# B&R Automation Studio project Panasonic_LinkaPowerCP2_A2021055 (part 44)

#### Main.st - Init, cyclic, exit code
```iecst
PROGRAM _INIT
	(* Insert code here *)
	SKTcpClientTrace_1.Params.IPportClient := 19000;
	SKTcpClientTrace_1.Cmd.LoggerOn:= FALSE;
END_PROGRAM

PROGRAM _CYCLIC

	//Priradenie indexu paletky//
    a:= P3_StoperSrobovania.PAR.CisloPaletky;
	P3_StoperSrobovania.PAR.CisloPaletky_STRING:= USINT_TO_STRING(a);

    //Parametre komunikácie//
    memcpy(ADR(SKTcpClientTrace_1.Params.IPaddrServ),ADR('192.168.128.250'),SIZEOF('192.168.128.250'));

    SKTcpClientTrace_1.Params.IPportServ := 12000;

	SKTcpClientTrace_1.pDevice := ADR('HDD_LOGGER');
	SKTcpClientTrace_1.pFile := ADR('logger_sktcpclienttrace_7.log');
    SKTcpClientTrace_1();

    //Parametre komunikácie//
    //Vstupy pre server//
    SKTcpClientTrace_1.Params.Packet.type := TRCB_P3_Srobovanie_ST7.INPUTS.TYP_Prikazu;
    SKTcpClientTrace_1.Params.Packet.workplace := TRCB_P3_Srobovanie_ST7.INPUTS.CisloStanice;
    SKTcpClientTrace_1.Params.Packet.rfid := TRCB_P3_Srobovanie_ST7.INPUTS.CisloPaletky;
    SKTcpClientTrace_1.Params.Packet.master := TRCB_P3_Srobovanie_ST7.INPUTS.QRkodPowerCP;
    SKTcpClientTrace_1.Params.Packet.dps1:= TRCB_P3_Srobovanie_ST7.INPUTS.QRkodFiltra;
    SKTcpClientTrace_1.Params.Packet.dps2:= '';
    SKTcpClientTrace_1.Params.Packet.dps3:= '';
    SKTcpClientTrace_1.Params.Packet.dps4:= '';
    SKTcpClientTrace_1.Params.Packet.dps5:= '';
    SKTcpClientTrace_1.Params.Packet.operator_id := TRCB_P3_Srobovanie_ST7.INPUTS.ID_Operatora;
    SKTcpClientTrace_1.Params.Packet.data_report:= TRCB_P3_Srobovanie_ST7.INPUTS.Report;
    SKTcpClientTrace_1.Params.Packet.result := TRCB_P3_Srobovanie_ST7.INPUTS.StavPaletky;

    //Výstupy zo servera//
    TRCB_P3_Srobovanie_ST7.OUTPUTS.TYP_Prikazu:= SKTcpClientTrace_1.Internal.Splitter.out[1];
    TRCB_P3_Srobovanie_ST7.OUTPUTS.CisloStanice:= SKTcpClientTrace_1.Internal.Splitter.out[2];
    TRCB_P3_Srobovanie_ST7.OUTPUTS.CisloPaletky:= SKTcpClientTrace_1.Internal.Splitter.out[3];
    IF TRCB_P3_Srobovanie_ST7.INPUTS.TYP_Prikazu = '0' THEN
        TRCB_P3_Srobovanie_ST7.OUTPUTS.CisloEtikety:= SKTcpClientTrace_1.Internal.Splitter.out[4];
    ELSE
        TRCB_P3_Srobovanie_ST7.OUTPUTS.QRkodPowerCP:= SKTcpClientTrace_1.Internal.Splitter.out[4];
    END_IF
    TRCB_P3_Srobovanie_ST7.OUTPUTS.QRkodFiltra:= SKTcpClientTrace_1.Internal.Splitter.out[5];
    TRCB_P3_Srobovanie_ST7.OUTPUTS.ID_Operatora:= SKTcpClientTrace_1.Internal.Splitter.out[10];
    TRCB_P3_Srobovanie_ST7.OUTPUTS.DruhCinnostiNaPaletke:= SKTcpClientTrace_1.Internal.Splitter.out[11];
    TRCB_P3_Srobovanie_ST7.OUTPUTS.PovolenieCinnostiNaPaletke:= SKTcpClientTrace_1.Internal.Splitter.out[12];

    //Volanie funkcie SequenceControl//
    SequenceControl(SC:= SC_KOM_Server);

    CASE SC_KOM_Server.Step OF

        0:
            SC_KOM_Server.StepName:= '0 - Nulovanie';
            SKTcpClientTrace_1.Cmd.Send:= FALSE;
            TRCB_P3_Srobovanie_ST7.CMD.VyziadajStavPaletky_TYP1:= FALSE;
            TRCB_P3_Srobovanie_ST7.CMD.PriradQRkodFiltra_TYP3:= FALSE;
            TRCB_P3_Srobovanie_ST7.CMD.VyziadajCisloEtikety_TYP0:= FALSE;
            TRCB_P3_Srobovanie_ST7.CMD.OdosliStavPaletky_TYP2:= FALSE;
            TRCB_P3_Srobovanie_ST7.STATUS.KomunikaciaUkoncena:= FALSE;
			TRCB_P3_Srobovanie_ST7.STATUS.KomunikaciaError:= FALSE;
			TRCB_P3_Srobovanie_ST7.STATUS.KOM_READY:= FALSE;
            PocetDopytovNaServer:= 0;

            IF SKTcpClientTrace_1.Internal.Step = 0 THEN
                SKTcpClientTrace_1.Enable:= TRUE;
                SC_KOM_Server.ResetStep:= TRUE;
                SC_KOM_Server.Step:= 1;
            ELSIF SKTcpClientTrace_1.Internal.Step = 15 THEN
                SKTcpClientTrace_1.Enable:= TRUE;
                SC_KOM_Server.ResetStep:= TRUE;
                SC_KOM_Server.Step:= 1;
            ELSE
                SKTcpClientTrace_1.Enable:= FALSE;
            END_IF

        1:
            SC_KOM_Server.StepName:= '1 - Rozhodnutie o cinnosti';
            TRCB_P3_Srobovanie_ST7.STATUS.KOM_READY:= TRUE;
			IF TRCB_P3_Srobovanie_ST7.CMD.VyziadajStavPaletky_TYP1 THEN
                TRCB_P3_Srobovanie_ST7.STATUS.KOM_READY:= FALSE;
				SC_KOM_Server.Step:= 10;
            ELSIF TRCB_P3_Srobovanie_ST7.CMD.PriradQRkodFiltra_TYP3 THEN
                TRCB_P3_Srobovanie_ST7.STATUS.KOM_READY:= FALSE;
				SC_KOM_Server.Step:= 20;
            ELSIF TRCB_P3_Srobovanie_ST7.CMD.VyziadajCisloEtikety_TYP0 THEN
                TRCB_P3_Srobovanie_ST7.STATUS.KOM_READY:= FALSE;
				SC_KOM_Server.Step:= 30;
            ELSIF TRCB_P3_Srobovanie_ST7.CMD.OdosliStavPaletky_TYP2 THEN
				TRCB_P3_Srobovanie_ST7.STATUS.KOM_READY:= FALSE;
				SC_KOM_Server.Step:= 40;
			ELSIF TRCB_P3_Srobovanie_ST7.CMD.VyziadajStavPanatrace_TYP4 THEN
				TRCB_P3_Srobovanie_ST7.STATUS.KOM_READY:= FALSE;
				SC_KOM_Server.Step:= 50;
            END_IF

        10:
            SC_KOM_Server.StepName:= '10 - Vyziadanie stavu paletky - odoslanie dat na server';
            SC_KOM_Server.IdleTime.PT:= T#3s;
            SC_KOM_Server.AlarmTime.PT:= T#10s;
            SC_KOM_Server.AlarmTime.IN:= TRUE;

			TRCB_P3_Srobovanie_ST7.INPUTS.CisloPaletky:= 'Pal';
			brsstrcat(ADR(TRCB_P3_Srobovanie_ST7.INPUTS.CisloPaletky), ADR(P3_StoperSrobovania.PAR.CisloPaletky_STRING));

            TRCB_P3_Srobovanie_ST7.INPUTS.TYP_Prikazu:= '1';
            TRCB_P3_Srobovanie_ST7.INPUTS.CisloStanice:= 'ST7';
            TRCB_P3_Srobovanie_ST7.INPUTS.QRkodPowerCP:= Paletka[a].PAR.QRkodPowerCP;
            TRCB_P3_Srobovanie_ST7.INPUTS.QRkodFiltra:= '';
            TRCB_P3_Srobovanie_ST7.INPUTS.ID_Operatora:= Paletka[a].PAR.ID_Operatora;
            TRCB_P3_Srobovanie_ST7.INPUTS.Report:= '';
            TRCB_P3_Srobovanie_ST7.INPUTS.StavPaletky:= 'OK';

			IF SKTcpClientTrace_1.Status.staReadyToSend AND NOT SKTcpClientTrace_1.Cmd.Close THEN
				TRCB_P3_Srobovanie_ST7.OUTPUTS.TYP_Prikazu:= '';
				SKTcpClientTrace_1.Cmd.Send:= TRUE;
				SC_KOM_Server.ResetStep:= TRUE;
				SC_KOM_Server.Step:= 13;
			END_IF

		13:
            SC_KOM_Server.StepName:= '13 - Vyziadanie stavu paletky - odpoved servera';
            SC_KOM_Server.IdleTime.PT:= T#3s;
            SC_KOM_Server.AlarmTime.PT:= T#7s;
            SC_KOM_Server.AlarmTime.IN:= TRUE;

            IF SKTcpClientTrace_1.Status.staReceived AND
                (TRCB_P3_Srobovanie_ST7.OUTPUTS.TYP_Prikazu = TRCB_P3_Srobovanie_ST7.INPUTS.TYP_Prikazu) AND
                (TRCB_P3_Srobovanie_ST7.OUTPUTS.QRkodPowerCP = TRCB_P3_Srobovanie_ST7.INPUTS.QRkodPowerCP) THEN
                TRCB_P3_Srobovanie_ST7.STATUS.KomunikaciaUkoncena:= TRUE;
                SC_KOM_Server.ResetStep:= TRUE;
                SC_KOM_Server.Step:= 15;
            ELSIF SC_KOM_Server.AlarmTime.Q AND NOT SKTcpClientTrace_1.Status.staSending THEN
                PocetDopytovNaServer:= PocetDopytovNaServer + 1;
				SKTcpClientTrace_1.Cmd.Send:= FALSE;
				SKTcpClientTrace_1.Cmd.Close:= TRUE;
				SC_KOM_Server.ResetStep:= TRUE;
                SC_KOM_Server.Step:= 14;
            END_IF

        14:
            SC_KOM_Server.StepName:= '14 - Vyziadanie stavu paletky - cakam na opatovny dopyt na server';
            SC_KOM_Server.IdleTime.PT:= T#1s;
            SC_KOM_Server.AlarmTime.PT:= T#10s;
            SC_KOM_Server.IdleTime.IN:= TRUE;

            IF PocetDopytovNaServer < 3 THEN
                IF SC_KOM_Server.IdleTime.Q THEN
                    SC_KOM_Server.ResetStep:= TRUE;
                    SC_KOM_Server.Step:= 10;
                END_IF
            ELSE
                TRCB_P3_Srobovanie_ST7.STATUS.KomunikaciaError:= TRUE;
                SC_KOM_Server.ResetStep:= TRUE;
                SC_KOM_Server.Step:= 15;
            END_IF

        15:
            SC_KOM_Server.StepName:= '15 - Vyziadanie stavu paletky - cakam na ukoncenie komunikacie';
            SC_KOM_Server.IdleTime.PT:= T#3s;
            SC_KOM_Server.AlarmTime.PT:= T#10s;

            IF NOT TRCB_P3_Srobovanie_ST7.CMD.VyziadajStavPaletky_TYP1 THEN
                SC_KOM_Server.ResetStep:= TRUE;
                SC_KOM_Server.Step:= 0;
            END_IF

        20:
            SC_KOM_Server.StepName:= '20 - Priradenie QR kodu - odoslanie dat na server';
            SC_KOM_Server.IdleTime.PT:= T#3s;
            SC_KOM_Server.AlarmTime.PT:= T#10s;

            TRCB_P3_Srobovanie_ST7.INPUTS.TYP_Prikazu:= '3';
            TRCB_P3_Srobovanie_ST7.INPUTS.CisloStanice:= 'ST7';
            TRCB_P3_Srobovanie_ST7.INPUTS.CisloPaletky;
            TRCB_P3_Srobovanie_ST7.INPUTS.QRkodPowerCP:= Paletka[a].PAR.QRkodPowerCP;
            TRCB_P3_Srobovanie_ST7.INPUTS.QRkodFiltra:= '';
            TRCB_P3_Srobovanie_ST7.INPUTS.ID_Operatora:= Paletka[a].PAR.ID_Operatora;
            TRCB_P3_Srobovanie_ST7.INPUTS.Report:= '';
            TRCB_P3_Srobovanie_ST7.INPUTS.StavPaletky:= 'OK';
            SKTcpClientTrace_1.Cmd.Send:= TRUE;

            IF SKTcpClientTrace_1.Cmd.Send AND NOT SKTcpClientTrace_1.Status.staReceived AND NOT SKTcpClientTrace_1.Status.staError THEN
                SC_KOM_Server.ResetStep:= TRUE;
                SC_KOM_Server.Step:= 23;
            END_IF

        23:
            SC_KOM_Server.StepName:= '23 - Priradenie QR kodu - odpoved servera';
            SC_KOM_Server.IdleTime.PT:= T#3s;
            SC_KOM_Server.AlarmTime.PT:= T#20s;
            SC_KOM_Server.AlarmTime.IN:= TRUE;

            IF SKTcpClientTrace_1.Status.staReceived AND
                (TRCB_P3_Srobovanie_ST7.OUTPUTS.TYP_Prikazu = TRCB_P3_Srobovanie_ST7.INPUTS.TYP_Prikazu) AND
                (TRCB_P3_Srobovanie_ST7.OUTPUTS.QRkodPowerCP = TRCB_P3_Srobovanie_ST7.INPUTS.QRkodPowerCP) THEN
                TRCB_P3_Srobovanie_ST7.STATUS.KomunikaciaUkoncena:= TRUE;
                SC_KOM_Server.ResetStep:= TRUE;
                SC_KOM_Server.Step:= 25;
            ELSIF SC_KOM_Server.AlarmTime.Q THEN
                TRCB_P3_Srobovanie_ST7.STATUS.KomunikaciaError:= TRUE;
                SC_KOM_Server.ResetStep:= TRUE;
                SC_KOM_Server.Step:= 25;
            END_IF

        25:
            SC_KOM_Server.StepName:= '25 - Vyziadanie stavu paletky - cakam na ukoncenie komunikacie';
            SC_KOM_Server.IdleTime.PT:= T#3s;
            SC_KOM_Server.AlarmTime.PT:= T#10s;

            IF NOT TRCB_P3_Srobovanie_ST7.CMD.PriradQRkodFiltra_TYP3 THEN
                SC_KOM_Server.ResetStep:= TRUE;
                SC_KOM_Server.Step:= 0;
            END_IF

        30:
            SC_KOM_Server.StepName:= '30 - Vyziadanie serioveho cisla - odoslanie dat na server';
            SC_KOM_Server.IdleTime.PT:= T#3s;
            SC_KOM_Server.AlarmTime.PT:= T#10s;

            TRCB_P3_Srobovanie_ST7.INPUTS.TYP_Prikazu:= '0';
            TRCB_P3_Srobovanie_ST7.INPUTS.CisloStanice:= 'ST7';
            TRCB_P3_Srobovanie_ST7.INPUTS.CisloPaletky;
            TRCB_P3_Srobovanie_ST7.INPUTS.QRkodPowerCP:= '';
            TRCB_P3_Srobovanie_ST7.INPUTS.QRkodFiltra:= '';
            TRCB_P3_Srobovanie_ST7.INPUTS.ID_Operatora:= 'E2';
            TRCB_P3_Srobovanie_ST7.INPUTS.Report:= '';
            TRCB_P3_Srobovanie_ST7.INPUTS.StavPaletky:= 'OK';
            SKTcpClientTrace_1.Cmd.Send:= TRUE;

            IF SKTcpClientTrace_1.Cmd.Send AND NOT SKTcpClientTrace_1.Status.staReceived AND NOT SKTcpClientTrace_1.Status.staError THEN
                SC_KOM_Server.ResetStep:= TRUE;
                SC_KOM_Server.Step:= 33;
            END_IF

        33:
            SC_KOM_Server.StepName:= '33 - Vyziadanie serioveho cisla - odpoved servera';
            SC_KOM_Server.IdleTime.PT:= T#3s;
            SC_KOM_Server.AlarmTime.PT:= T#20s;
            SC_KOM_Server.AlarmTime.IN:= TRUE;

            IF SKTcpClientTrace_1.Status.staReceived AND
                (TRCB_P3_Srobovanie_ST7.OUTPUTS.TYP_Prikazu = TRCB_P3_Srobovanie_ST7.INPUTS.TYP_Prikazu) THEN
                TRCB_P3_Srobovanie_ST7.STATUS.KomunikaciaUkoncena:= TRUE;
                SC_KOM_Server.ResetStep:= TRUE;
                SC_KOM_Server.Step:= 35;
            ELSIF SC_KOM_Server.AlarmTime.Q THEN
                TRCB_P3_Srobovanie_ST7.STATUS.KomunikaciaError:= TRUE;
                SC_KOM_Server.ResetStep:= TRUE;
                SC_KOM_Server.Step:= 35;
            END_IF

        35:
            SC_KOM_Server.StepName:= '35 - Vyziadanie serioveho cisla - cakam na ukoncenie komunikacie';
            SC_KOM_Server.IdleTime.PT:= T#3s;
            SC_KOM_Server.AlarmTime.PT:= T#10s;

            IF NOT TRCB_P3_Srobovanie_ST7.CMD.VyziadajCisloEtikety_TYP0 THEN
                SC_KOM_Server.ResetStep:= TRUE;
                SC_KOM_Server.Step:= 0;
            END_IF

        40:
            SC_KOM_Server.StepName:= '40 - Odoslanie stavu paletky - odoslanie dat na server';
            SC_KOM_Server.IdleTime.PT:= T#3s;
            SC_KOM_Server.AlarmTime.PT:= T#20s;
            SC_KOM_Server.AlarmTime.IN:= TRUE;

            //Vytvorenie spravy pre report//
            IF NOT SC_KOM_Server.Switch1 THEN
                brsmemset(ADR(Report),0,SIZEOF(Report));
                brsmemset(ADR(TRCB_P3_Srobovanie_ST7.INPUTS.Report), 0, SIZEOF(TRCB_P3_Srobovanie_ST7.INPUTS.Report));

				//Skrutka K40//
                Report[0].PoradoveCislo:= '1';
                Report[0].Popis:= 'SkrutkaK40_Moment';
                Report[0].FormatHodnoty:= '1';
                Report[0].Tolerancia_MIN_Hodnota:= Reports.Skrutkovacky.Moment_ToleranciaMIN.P3_SkrutkaK40;
                Report[0].Tolerancia_MAX_Hodnota:= Reports.Skrutkovacky.Moment_ToleranciaMAX.P3_SkrutkaK40;
                Report[0].Nominal:= '';
                Report[0].Tolerancia_MIN_Jednotky:= 'Nm';
                Report[0].Tolerancia_MAX_Jednotky:= 'Nm';
                Report[0].NameranaHodnota:= Reports.Skrutkovacky.Moment_NameranaHodnota.P3_SkrutkaK40;
                Report[0].NameranaHodnota_Jednotky:= 'Nm';
                Report[0].VyslednyResult:= Reports.Skrutkovacky.VyslednyReport.P3_SkrutkaK40;
                SKTcpClientNewCsvEntry(Report[0].PoradoveCislo,Report[0].Popis,Report[0].FormatHodnoty,Report[0].Tolerancia_MIN_Hodnota,Report[0].Tolerancia_MAX_Hodnota,Report[0].Nominal,Report[0].Tolerancia_MIN_Jednotky,Report[0].Tolerancia_MAX_Jednotky,Report[0].NameranaHodnota,Report[0].NameranaHodnota_Jednotky,Report[0].VyslednyResult, ADR(TRCB_P3_Srobovanie_ST7.INPUTS.Report));

                Report[1].PoradoveCislo:= '2';
                Report[1].Popis:= 'SkrutkaK40_Uhol';
                Report[1].FormatHodnoty:= '1';
                Report[1].Tolerancia_MIN_Hodnota:= Reports.Skrutkovacky.Uhol_ToleranciaMIN.P3_SkrutkaK40;
                Report[1].Tolerancia_MAX_Hodnota:= Reports.Skrutkovacky.Uhol_ToleranciaMAX.P3_SkrutkaK40;
                Report[1].Nominal:= '';
                Report[1].Tolerancia_MIN_Jednotky:= 'st';
                Report[1].Tolerancia_MAX_Jednotky:= 'st';
                Report[1].NameranaHodnota:= Reports.Skrutkovacky.Uhol_NameranaHodnota.P3_SkrutkaK40;
                Report[1].NameranaHodnota_Jednotky:= 'st';
                Report[1].VyslednyResult:= Reports.Skrutkovacky.VyslednyReport.P3_SkrutkaK40;
                SKTcpClientNewCsvEntry(Report[1].PoradoveCislo,Report[1].Popis,Report[1].FormatHodnoty,Report[1].Tolerancia_MIN_Hodnota,Report[1].Tolerancia_MAX_Hodnota,Report[1].Nominal,Report[1].Tolerancia_MIN_Jednotky,Report[1].Tolerancia_MAX_Jednotky,Report[1].NameranaHodnota,Report[1].NameranaHodnota_Jednotky,Report[1].VyslednyResult, ADR(TRCB_P3_Srobovanie_ST7.INPUTS.Report));

                Report[2].PoradoveCislo:= '3';
                Report[2].Popis:= 'SkrutkaK40_CasSrobovania';
                Report[2].FormatHodnoty:= '1';
                Report[2].Tolerancia_MIN_Hodnota:= '';
                Report[2].Tolerancia_MAX_Hodnota:= '';
                Report[2].Nominal:= '';
                Report[2].Tolerancia_MIN_Jednotky:= '';
                Report[2].Tolerancia_MAX_Jednotky:= '';
                Report[2].NameranaHodnota:= Reports.Skrutkovacky.CasSkrutkovania.P3_SkrutkaK40;
                Report[2].NameranaHodnota_Jednotky:= 's';
                Report[2].VyslednyResult:= Reports.Skrutkovacky.VyslednyReport.P3_SkrutkaK40;
                SKTcpClientNewCsvEntry(Report[2].PoradoveCislo,Report[2].Popis,Report[2].FormatHodnoty,Report[2].Tolerancia_MIN_Hodnota,Report[2].Tolerancia_MAX_Hodnota,Report[2].Nominal,Report[2].Tolerancia_MIN_Jednotky,Report[2].Tolerancia_MAX_Jednotky,Report[2].NameranaHodnota,Report[2].NameranaHodnota_Jednotky,Report[2].VyslednyResult, ADR(TRCB_P3_Srobovanie_ST7.INPUTS.Report));

                Report[3].PoradoveCislo:= '4';
                Report[3].Popis:= 'SkrutkaK40_VyskaSrobovania';
                Report[3].FormatHodnoty:= '1';
                Report[3].Tolerancia_MIN_Hodnota:= '';
                Report[3].Tolerancia_MAX_Hodnota:= '';
                Report[3].Nominal:= '';
                Report[3].Tolerancia_MIN_Jednotky:= '';
                Report[3].Tolerancia_MAX_Jednotky:= '';
                Report[3].NameranaHodnota:= Reports.Skrutkovacky.VyskaSkrutkovania.P3_SkrutkaK40;
                Report[3].NameranaHodnota_Jednotky:= 'mm';
                Report[3].VyslednyResult:= Reports.Skrutkovacky.VyslednyReport.P3_SkrutkaK40;
                SKTcpClientNewCsvEntry(Report[3].PoradoveCislo,Report[3].Popis,Report[3].FormatHodnoty,Report[3].Tolerancia_MIN_Hodnota,Report[3].Tolerancia_MAX_Hodnota,Report[3].Nominal,Report[3].Tolerancia_MIN_Jednotky,Report[3].Tolerancia_MAX_Jednotky,Report[3].NameranaHodnota,Report[3].NameranaHodnota_Jednotky,Report[3].VyslednyResult, ADR(TRCB_P3_Srobovanie_ST7.INPUTS.Report));

                //Skrutka M5//
                Report[4].PoradoveCislo:= '5';
                Report[4].Popis:= 'SkrutkaM5_Moment';
                Report[4].FormatHodnoty:= '1';
                Report[4].Tolerancia_MIN_Hodnota:= Reports.Skrutkovacky.Moment_ToleranciaMIN.P3_SkrutkaM5;
                Report[4].Tolerancia_MAX_Hodnota:= Reports.Skrutkovacky.Moment_ToleranciaMAX.P3_SkrutkaM5;
                Report[4].Nominal:= '';
                Report[4].Tolerancia_MIN_Jednotky:= 'Nm';
                Report[4].Tolerancia_MAX_Jednotky:= 'Nm';
                Report[4].NameranaHodnota:= Reports.Skrutkovacky.Moment_NameranaHodnota.P3_SkrutkaM5;
                Report[4].NameranaHodnota_Jednotky:= 'Nm';
                Report[4].VyslednyResult:= Reports.Skrutkovacky.VyslednyReport.P3_SkrutkaM5;
                SKTcpClientNewCsvEntry(Report[4].PoradoveCislo,Report[4].Popis,Report[4].FormatHodnoty,Report[4].Tolerancia_MIN_Hodnota,Report[4].Tolerancia_MAX_Hodnota,Report[4].Nominal,Report[4].Tolerancia_MIN_Jednotky,Report[4].Tolerancia_MAX_Jednotky,Report[4].NameranaHodnota,Report[4].NameranaHodnota_Jednotky,Report[4].VyslednyResult, ADR(TRCB_P3_Srobovanie_ST7.INPUTS.Report));

                Report[5].PoradoveCislo:= '6';
                Report[5].Popis:= 'SkrutkaM5_Uhol';
                Report[5].FormatHodnoty:= '1';
                Report[5].Tolerancia_MIN_Hodnota:= Reports.Skrutkovacky.Uhol_ToleranciaMIN.P3_SkrutkaM5;
                Report[5].Tolerancia_MAX_Hodnota:= Reports.Skrutkovacky.Uhol_ToleranciaMAX.P3_SkrutkaM5;
                Report[5].Nominal:= '';
                Report[5].Tolerancia_MIN_Jednotky:= 'st';
                Report[5].Tolerancia_MAX_Jednotky:= 'st';
                Report[5].NameranaHodnota:= Reports.Skrutkovacky.Uhol_NameranaHodnota.P3_SkrutkaM5;
                Report[5].NameranaHodnota_Jednotky:= 'st';
                Report[5].VyslednyResult:= Reports.Skrutkovacky.VyslednyReport.P3_SkrutkaM5;
                SKTcpClientNewCsvEntry(Report[5].PoradoveCislo,Report[5].Popis,Report[5].FormatHodnoty,Report[5].Tolerancia_MIN_Hodnota,Report[5].Tolerancia_MAX_Hodnota,Report[5].Nominal,Report[5].Tolerancia_MIN_Jednotky,Report[5].Tolerancia_MAX_Jednotky,Report[5].NameranaHodnota,Report[5].NameranaHodnota_Jednotky,Report[5].VyslednyResult, ADR(TRCB_P3_Srobovanie_ST7.INPUTS.Report));

                Report[6].PoradoveCislo:= '7';
                Report[6].Popis:= 'SkrutkaM5_CasSrobovania';
                Report[6].FormatHodnoty:= '1';
                Report[6].Tolerancia_MIN_Hodnota:= '';
                Report[6].Tolerancia_MAX_Hodnota:= '';
                Report[6].Nominal:= '';
                Report[6].Tolerancia_MIN_Jednotky:= '';
                Report[6].Tolerancia_MAX_Jednotky:= '';
                Report[6].NameranaHodnota:= Reports.Skrutkovacky.CasSkrutkovania.P3_SkrutkaM5;
                Report[6].NameranaHodnota_Jednotky:= 's';
                Report[6].VyslednyResult:= Reports.Skrutkovacky.VyslednyReport.P3_SkrutkaM5;
                SKTcpClientNewCsvEntry(Report[6].PoradoveCislo,Report[6].Popis,Report[6].FormatHodnoty,Report[6].Tolerancia_MIN_Hodnota,Report[6].Tolerancia_MAX_Hodnota,Report[6].Nominal,Report[6].Tolerancia_MIN_Jednotky,Report[6].Tolerancia_MAX_Jednotky,Report[6].NameranaHodnota,Report[6].NameranaHodnota_Jednotky,Report[6].VyslednyResult, ADR(TRCB_P3_Srobovanie_ST7.INPUTS.Report));

                Report[7].PoradoveCislo:= '8';
                Report[7].Popis:= 'SkrutkaM5_VyskaSrobovania';
                Report[7].FormatHodnoty:= '1';
                Report[7].Tolerancia_MIN_Hodnota:= '';
                Report[7].Tolerancia_MAX_Hodnota:= '';
                Report[7].Nominal:= '';
                Report[7].Tolerancia_MIN_Jednotky:= '';
                Report[7].Tolerancia_MAX_Jednotky:= '';
                Report[7].NameranaHodnota:= Reports.Skrutkovacky.VyskaSkrutkovania.P3_SkrutkaM5;
                Report[7].NameranaHodnota_Jednotky:= 'mm';
                Report[7].VyslednyResult:= Reports.Skrutkovacky.VyslednyReport.P3_SkrutkaM5;
                SKTcpClientNewCsvEntry(Report[7].PoradoveCislo,Report[7].Popis,Report[7].FormatHodnoty,Report[7].Tolerancia_MIN_Hodnota,Report[7].Tolerancia_MAX_Hodnota,Report[7].Nominal,Report[7].Tolerancia_MIN_Jednotky,Report[7].Tolerancia_MAX_Jednotky,Report[7].NameranaHodnota,Report[7].NameranaHodnota_Jednotky,Report[7].VyslednyResult, ADR(TRCB_P3_Srobovanie_ST7.INPUTS.Report));

//                //Kamera 13//
//                Report[8].PoradoveCislo:= '9';
//                Report[8].Popis:= 'KAM_13_KontrolaPaletky';
//                Report[8].FormatHodnoty:= '2';
//                Report[8].Tolerancia_MIN_Hodnota:= '';
//                Report[8].Tolerancia_MAX_Hodnota:= '';
//                Report[8].Nominal:= 'OK';
//                Report[8].Tolerancia_MIN_Jednotky:= '';
//                Report[8].Tolerancia_MAX_Jednotky:= '';
//                IF Reports.Kamery.P3_CAM13_KontrolaPaletky = 'PASS' THEN
//                    Report[8].NameranaHodnota:= 'OK';
//                ELSE
//                    Report[8].NameranaHodnota:= 'NG';
//                END_IF
//                Report[8].NameranaHodnota_Jednotky:= '';
//                Report[8].VyslednyResult:= Reports.Kamery.P3_CAM13_KontrolaPaletky;
//                SKTcpClientNewCsvEntry(Report[8].PoradoveCislo,Report[8].Popis,Report[8].FormatHodnoty,Report[8].Tolerancia_MIN_Hodnota,Report[8].Tolerancia_MAX_Hodnota,Report[8].Nominal,Report[8].Tolerancia_MIN_Jednotky,Report[8].Tolerancia_MAX_Jednotky,Report[8].NameranaHodnota,Report[8].NameranaHodnota_Jednotky,Report[8].VyslednyResult, ADR(TRCB_P3_Srobovanie_ST7.INPUTS.Report));
//
                SC_KOM_Server.Switch1:= TRUE;
            END_IF

			TRCB_P3_Srobovanie_ST7.INPUTS.CisloPaletky:= 'Pal';
			brsstrcat(ADR(TRCB_P3_Srobovanie_ST7.INPUTS.CisloPaletky), ADR(P3_StoperSrobovania.PAR.CisloPaletky_STRING));

            TRCB_P3_Srobovanie_ST7.INPUTS.TYP_Prikazu:= '2';
            TRCB_P3_Srobovanie_ST7.INPUTS.CisloStanice:= 'ST7';
            TRCB_P3_Srobovanie_ST7.INPUTS.QRkodPowerCP:= Paletka[a].PAR.QRkodPowerCP;
            TRCB_P3_Srobovanie_ST7.INPUTS.QRkodFiltra:= '';
            TRCB_P3_Srobovanie_ST7.INPUTS.ID_Operatora:= Paletka[a].PAR.ID_Operatora;
            TRCB_P3_Srobovanie_ST7.INPUTS.StavPaletky:= Paletka[a].PAR.StavPowerCP;

			IF SKTcpClientTrace_1.Status.staReadyToSend AND NOT SKTcpClientTrace_1.Cmd.Close THEN
				TRCB_P3_Srobovanie_ST7.OUTPUTS.TYP_Prikazu:= '';
				SKTcpClientTrace_1.Cmd.Send:= TRUE;
				SC_KOM_Server.ResetStep:= TRUE;
				SC_KOM_Server.Step:= 43;
			END_IF

        43:
            SC_KOM_Server.StepName:= '43 - Odoslanie stavu paletky - odpoved servera';
			SC_KOM_Server.IdleTime.PT:= T#3s;
            SC_KOM_Server.AlarmTime.PT:= T#7s;
            SC_KOM_Server.AlarmTime.IN:= TRUE;

            IF SKTcpClientTrace_1.Status.staReceived AND
                (TRCB_P3_Srobovanie_ST7.OUTPUTS.TYP_Prikazu = TRCB_P3_Srobovanie_ST7.INPUTS.TYP_Prikazu) AND
                (TRCB_P3_Srobovanie_ST7.OUTPUTS.QRkodPowerCP = TRCB_P3_Srobovanie_ST7.INPUTS.QRkodPowerCP) THEN
                TRCB_P3_Srobovanie_ST7.STATUS.KomunikaciaUkoncena:= TRUE;
                SC_KOM_Server.ResetStep:= TRUE;
                SC_KOM_Server.Step:= 45;
            ELSIF SC_KOM_Server.AlarmTime.Q AND NOT SKTcpClientTrace_1.Status.staSending THEN
                PocetDopytovNaServer:= PocetDopytovNaServer + 1;
				SKTcpClientTrace_1.Cmd.Send:= FALSE;
				SKTcpClientTrace_1.Cmd.Close:= TRUE;
				SC_KOM_Server.ResetStep:= TRUE;
                SC_KOM_Server.Step:= 44;
            END_IF

        44:
            SC_KOM_Server.StepName:= '44 - Odoslanie stavu paletky - cakam na opatovny dopyt na server';
            SC_KOM_Server.IdleTime.PT:= T#1s;
            SC_KOM_Server.AlarmTime.PT:= T#10s;
            SC_KOM_Server.IdleTime.IN:= TRUE;
            SKTcpClientTrace_1.Cmd.Send:= FALSE;

            IF PocetDopytovNaServer < 3 THEN
                IF SC_KOM_Server.IdleTime.Q THEN
                    SC_KOM_Server.ResetStep:= TRUE;
                    SC_KOM_Server.Step:= 40;
                END_IF
            ELSE
                TRCB_P3_Srobovanie_ST7.STATUS.KomunikaciaError:= TRUE;
                SC_KOM_Server.ResetStep:= TRUE;
                SC_KOM_Server.Step:= 45;
            END_IF

        45:
            SC_KOM_Server.StepName:= '45 - Vyziadanie serioveho cisla - cakam na ukoncenie komunikacie';
            SC_KOM_Server.IdleTime.PT:= T#3s;
            SC_KOM_Server.AlarmTime.PT:= T#10s;

            IF NOT TRCB_P3_Srobovanie_ST7.CMD.OdosliStavPaletky_TYP2 THEN
                SC_KOM_Server.ResetStep:= TRUE;
                SC_KOM_Server.Step:= 0;
            END_IF

		50:
			SC_KOM_Server.StepName:= '50 - Vyziadanie stavu Panatrace - odoslanie dat na server';
			SC_KOM_Server.IdleTime.PT:= T#3s;
			SC_KOM_Server.AlarmTime.PT:= T#10s;
			SC_KOM_Server.AlarmTime.IN:= TRUE;

			TRCB_P3_Srobovanie_ST7.INPUTS.TYP_Prikazu:= '4';
			TRCB_P3_Srobovanie_ST7.INPUTS.CisloStanice:= 'ST7';
			TRCB_P3_Srobovanie_ST7.INPUTS.CisloPaletky:= '';
			TRCB_P3_Srobovanie_ST7.INPUTS.QRkodPowerCP:= '';
			TRCB_P3_Srobovanie_ST7.INPUTS.QRkodFiltra:= '';
			TRCB_P3_Srobovanie_ST7.INPUTS.ID_Operatora:= '';
			TRCB_P3_Srobovanie_ST7.INPUTS.Report:= '';
			TRCB_P3_Srobovanie_ST7.INPUTS.StavPaletky:= '';

			IF SKTcpClientTrace_1.Status.staReadyToSend AND NOT SKTcpClientTrace_1.Cmd.Close THEN
				TRCB_P3_Srobovanie_ST7.OUTPUTS.TYP_Prikazu:= '';
				SKTcpClientTrace_1.Cmd.Send:= TRUE;
				SC_KOM_Server.ResetStep:= TRUE;
				SC_KOM_Server.Step:= 53;
			END_IF

		53:
			SC_KOM_Server.StepName:= '53 - Vyziadanie stavu paletky - odpoved servera';
			SC_KOM_Server.IdleTime.PT:= T#30s;
			SC_KOM_Server.AlarmTime.PT:= T#7s;
			SC_KOM_Server.AlarmTime.IN:= TRUE;

			IF SKTcpClientTrace_1.Status.staReceived AND TRCB_P3_Srobovanie_ST7.OUTPUTS.TYP_Prikazu = TRCB_P3_Srobovanie_ST7.INPUTS.TYP_Prikazu THEN
				TRCB_P3_Srobovanie_ST7.STATUS.KomunikaciaUkoncena:= TRUE;
				SC_KOM_Server.ResetStep:= TRUE;
				SC_KOM_Server.Step:= 55;
			ELSIF SC_KOM_Server.AlarmTime.Q AND NOT SKTcpClientTrace_1.Status.staSending THEN
				PocetDopytovNaServer:= PocetDopytovNaServer + 1;
				SKTcpClientTrace_1.Cmd.Send:= FALSE;
				SKTcpClientTrace_1.Cmd.Close:= TRUE;
				SC_KOM_Server.ResetStep:= TRUE;
				SC_KOM_Server.Step:= 54;
			END_IF

		54:
			SC_KOM_Server.StepName:= '54 - Vyziadanie stavu paletky - cakam na opatovny dopyt na server';
			SC_KOM_Server.IdleTime.PT:= T#1s;
			SC_KOM_Server.AlarmTime.PT:= T#10s;
			SC_KOM_Server.IdleTime.IN:= TRUE;

			IF PocetDopytovNaServer < 3 THEN
				IF SC_KOM_Server.IdleTime.Q THEN
					SC_KOM_Server.ResetStep:= TRUE;
					SC_KOM_Server.Step:= 50;
				END_IF
			ELSE
				TRCB_P3_Srobovanie_ST7.STATUS.KomunikaciaError:= TRUE;
				SC_KOM_Server.ResetStep:= TRUE;
				SC_KOM_Server.Step:= 55;
			END_IF

		55:
			SC_KOM_Server.StepName:= '55 - Vyziadanie stavu paletky - cakam na ukoncenie komunikacie';
			SC_KOM_Server.IdleTime.PT:= T#3s;
			SC_KOM_Server.AlarmTime.PT:= T#10s;

			IF NOT TRCB_P3_Srobovanie_ST7.CMD.VyziadajStavPanatrace_TYP4 THEN
				SC_KOM_Server.ResetStep:= TRUE;
				SC_KOM_Server.Step:= 0;
			END_IF

    END_CASE

END_PROGRAM

PROGRAM _EXIT
	(* Insert code here *)

END_PROGRAM
```

#### Types.typ - Local data types
```iecst
TYPE
	Report_typ : 	STRUCT
		PoradoveCislo : STRING[2]; (*IDstep - Poradové čislo reportu*)
		Popis : STRING[100]; (*Description - Popis*)
		FormatHodnoty : STRING[2]; (*TypValue - Format zaslané hodnoty  1- Číslo, 2 - Znak*)
		Tolerancia_MIN_Hodnota : STRING[10]; (*MinTol - Minimálna tolerancia meranej veličiny*)
		Tolerancia_MAX_Hodnota : STRING[10]; (*MaxTol - Maximálna tolerancia meranej veličiny*)
		Nominal : STRING[10]; (*Nom - Ak jezvolený formát string tak tu zadáme OK inak je prazdna*)
		Tolerancia_MIN_Jednotky : STRING[10]; (*MinEle - Jednotky minimálnej tolerancie veličiny*)
		Tolerancia_MAX_Jednotky : STRING[10]; (*MaxEle - Jednotky maximálnej tolerancie veličiny*)
		NameranaHodnota : STRING[10]; (*Value - Namerana hodnota veličiny, ak su kamery tak bude hodnota OK alebo NG*)
		NameranaHodnota_Jednotky : STRING[10]; (*ValEle - Jednotky nameranej veličiny*)
		VyslednyResult : STRING[5]; (*Result - Výsledný result  PASS, FAIL, SKIP*)
	END_STRUCT;
END_TYPE
```

#### Variables.var - Local variables
```iecst
VAR
	SC_KOM_Server : SequenceControlTyp;
	SKTcpClientTrace_1 : SKTcpClientTrace;
	a : USINT;
	Report : ARRAY[0..50] OF Report_typ;
	PocetDopytovNaServer : USINT;
END_VAR
```

### Program Logical/TracebilitySystem/P3_LeakageTestA_ST8A (IEC)

#### Main.st - Init, cyclic, exit code
```iecst
PROGRAM _INIT
	(* Insert code here *)
	SKTcpClientTrace_1.Params.IPportClient := 20000;
	SKTcpClientTrace_1.Cmd.LoggerOn:= FALSE;
END_PROGRAM

PROGRAM _CYCLIC

	//Priradenie indexu paletky//
    a:= P3_LeakageTestA.PAR.CisloPaletky;
	P3_LeakageTestA.PAR.CisloPaletky_STRING:= USINT_TO_STRING(a);

    //Parametre komunikácie//
    memcpy(ADR(SKTcpClientTrace_1.Params.IPaddrServ),ADR('192.168.128.250'),SIZEOF('192.168.128.250'));

    SKTcpClientTrace_1.Params.IPportServ := 12000;

	SKTcpClientTrace_1.pDevice := ADR('HDD_LOGGER');
	SKTcpClientTrace_1.pFile := ADR('logger_sktcpclienttrace_8A.log');
    SKTcpClientTrace_1();

    //Parametre komunikácie//
    //Vstupy pre server//
    SKTcpClientTrace_1.Params.Packet.type := TRCB_P3_LeakageTestA_ST8A.INPUTS.TYP_Prikazu;
    SKTcpClientTrace_1.Params.Packet.workplace := TRCB_P3_LeakageTestA_ST8A.INPUTS.CisloStanice;
    SKTcpClientTrace_1.Params.Packet.rfid := TRCB_P3_LeakageTestA_ST8A.INPUTS.CisloPaletky;
    SKTcpClientTrace_1.Params.Packet.master := TRCB_P3_LeakageTestA_ST8A.INPUTS.QRkodPowerCP;
    SKTcpClientTrace_1.Params.Packet.dps1:= TRCB_P3_LeakageTestA_ST8A.INPUTS.QRkodFiltra;
    SKTcpClientTrace_1.Params.Packet.dps2:= '';
    SKTcpClientTrace_1.Params.Packet.dps3:= '';
    SKTcpClientTrace_1.Params.Packet.dps4:= '';
    SKTcpClientTrace_1.Params.Packet.dps5:= '';
    SKTcpClientTrace_1.Params.Packet.operator_id := TRCB_P3_LeakageTestA_ST8A.INPUTS.ID_Operatora;
    SKTcpClientTrace_1.Params.Packet.data_report:= TRCB_P3_LeakageTestA_ST8A.INPUTS.Report;
    SKTcpClientTrace_1.Params.Packet.result := TRCB_P3_LeakageTestA_ST8A.INPUTS.StavPaletky;

    //Výstupy zo servera//
    TRCB_P3_LeakageTestA_ST8A.OUTPUTS.TYP_Prikazu:= SKTcpClientTrace_1.Internal.Splitter.out[1];
    TRCB_P3_LeakageTestA_ST8A.OUTPUTS.CisloStanice:= SKTcpClientTrace_1.Internal.Splitter.out[2];
    TRCB_P3_LeakageTestA_ST8A.OUTPUTS.CisloPaletky:= SKTcpClientTrace_1.Internal.Splitter.out[3];
    IF TRCB_P3_LeakageTestA_ST8A.INPUTS.TYP_Prikazu = '0' THEN
        TRCB_P3_LeakageTestA_ST8A.OUTPUTS.CisloEtikety:= SKTcpClientTrace_1.Internal.Splitter.out[4];
    ELSE
        TRCB_P3_LeakageTestA_ST8A.OUTPUTS.QRkodPowerCP:= SKTcpClientTrace_1.Internal.Splitter.out[4];
    END_IF
    TRCB_P3_LeakageTestA_ST8A.OUTPUTS.QRkodFiltra:= SKTcpClientTrace_1.Internal.Splitter.out[5];
    TRCB_P3_LeakageTestA_ST8A.OUTPUTS.ID_Operatora:= SKTcpClientTrace_1.Internal.Splitter.out[10];
    TRCB_P3_LeakageTestA_ST8A.OUTPUTS.DruhCinnostiNaPaletke:= SKTcpClientTrace_1.Internal.Splitter.out[11];
    TRCB_P3_LeakageTestA_ST8A.OUTPUTS.PovolenieCinnostiNaPaletke:= SKTcpClientTrace_1.Internal.Splitter.out[12];

    //Volanie funkcie SequenceControl//
    SequenceControl(SC:= SC_KOM_Server);

    CASE SC_KOM_Server.Step OF

        0:
            SC_KOM_Server.StepName:= '0 - Nulovanie';
            SKTcpClientTrace_1.Cmd.Send:= FALSE;
            TRCB_P3_LeakageTestA_ST8A.CMD.VyziadajStavPaletky_TYP1:= FALSE;
            TRCB_P3_LeakageTestA_ST8A.CMD.PriradQRkodFiltra_TYP3:= FALSE;
            TRCB_P3_LeakageTestA_ST8A.CMD.VyziadajCisloEtikety_TYP0:= FALSE;
			TRCB_P3_LeakageTestA_ST8A.CMD.OdosliStavPaletky_TYP2:= FALSE;
			TRCB_P3_LeakageTestA_ST8A.CMD.VyziadajStavPanatrace_TYP4:= FALSE;
            TRCB_P3_LeakageTestA_ST8A.STATUS.KomunikaciaUkoncena:= FALSE;
			TRCB_P3_LeakageTestA_ST8A.STATUS.KomunikaciaError:= FALSE;
			TRCB_P3_LeakageTestA_ST8A.STATUS.KOM_READY:= FALSE;
            PocetDopytovNaServer:= 0;

            IF SKTcpClientTrace_1.Internal.Step = 0 THEN
                SKTcpClientTrace_1.Enable:= TRUE;
                SC_KOM_Server.ResetStep:= TRUE;
                SC_KOM_Server.Step:= 1;
            ELSIF SKTcpClientTrace_1.Internal.Step = 15 THEN
                SKTcpClientTrace_1.Enable:= TRUE;
                SC_KOM_Server.ResetStep:= TRUE;
                SC_KOM_Server.Step:= 1;
            ELSE
                SKTcpClientTrace_1.Enable:= FALSE;
            END_IF

        1:
            SC_KOM_Server.StepName:= '1 - Rozhodnutie o cinnosti';
            TRCB_P3_LeakageTestA_ST8A.STATUS.KOM_READY:= TRUE;
			IF TRCB_P3_LeakageTestA_ST8A.CMD.VyziadajStavPaletky_TYP1 THEN
                TRCB_P3_LeakageTestA_ST8A.STATUS.KOM_READY:= FALSE;
				SC_KOM_Server.Step:= 10;
            ELSIF TRCB_P3_LeakageTestA_ST8A.CMD.PriradQRkodFiltra_TYP3 THEN
                TRCB_P3_LeakageTestA_ST8A.STATUS.KOM_READY:= FALSE;
				SC_KOM_Server.Step:= 20;
            ELSIF TRCB_P3_LeakageTestA_ST8A.CMD.VyziadajCisloEtikety_TYP0 THEN
                TRCB_P3_LeakageTestA_ST8A.STATUS.KOM_READY:= FALSE;
				SC_KOM_Server.Step:= 30;
            ELSIF TRCB_P3_LeakageTestA_ST8A.CMD.OdosliStavPaletky_TYP2 THEN
				TRCB_P3_LeakageTestA_ST8A.STATUS.KOM_READY:= FALSE;
				SC_KOM_Server.Step:= 40;
			ELSIF TRCB_P3_LeakageTestA_ST8A.CMD.VyziadajStavPanatrace_TYP4 THEN
				TRCB_P3_LeakageTestA_ST8A.STATUS.KOM_READY:= FALSE;
				SC_KOM_Server.Step:= 50;
            END_IF

        10:
            SC_KOM_Server.StepName:= '10 - Vyziadanie stavu paletky - odoslanie dat na server';
            SC_KOM_Server.IdleTime.PT:= T#3s;
            SC_KOM_Server.AlarmTime.PT:= T#10s;
            SC_KOM_Server.AlarmTime.IN:= TRUE;

			TRCB_P3_LeakageTestA_ST8A.INPUTS.CisloPaletky:= 'Pal';
			brsstrcat(ADR(TRCB_P3_LeakageTestA_ST8A.INPUTS.CisloPaletky), ADR(P3_LeakageTestA.PAR.CisloPaletky_STRING));

            TRCB_P3_LeakageTestA_ST8A.INPUTS.TYP_Prikazu:= '1';
            TRCB_P3_LeakageTestA_ST8A.INPUTS.CisloStanice:= 'ST8A';
            TRCB_P3_LeakageTestA_ST8A.INPUTS.QRkodPowerCP:= Paletka[a].PAR.QRkodPowerCP;
            TRCB_P3_LeakageTestA_ST8A.INPUTS.QRkodFiltra:= '';
            TRCB_P3_LeakageTestA_ST8A.INPUTS.ID_Operatora:= Paletka[a].PAR.ID_Operatora;
            TRCB_P3_LeakageTestA_ST8A.INPUTS.Report:= '';
            TRCB_P3_LeakageTestA_ST8A.INPUTS.StavPaletky:= 'OK';

			IF SKTcpClientTrace_1.Status.staReadyToSend AND NOT SKTcpClientTrace_1.Cmd.Close THEN
				TRCB_P3_LeakageTestA_ST8A.OUTPUTS.TYP_Prikazu:= '';
				SKTcpClientTrace_1.Cmd.Send:= TRUE;
				SC_KOM_Server.ResetStep:= TRUE;
				SC_KOM_Server.Step:= 13;
			END_IF

		13:
            SC_KOM_Server.StepName:= '13 - Vyziadanie stavu paletky - odpoved servera';
            SC_KOM_Server.IdleTime.PT:= T#3s;
            SC_KOM_Server.AlarmTime.PT:= T#7s;
            SC_KOM_Server.AlarmTime.IN:= TRUE;

            IF SKTcpClientTrace_1.Status.staReceived AND
                (TRCB_P3_LeakageTestA_ST8A.OUTPUTS.TYP_Prikazu = TRCB_P3_LeakageTestA_ST8A.INPUTS.TYP_Prikazu) AND
                (TRCB_P3_LeakageTestA_ST8A.OUTPUTS.QRkodPowerCP = TRCB_P3_LeakageTestA_ST8A.INPUTS.QRkodPowerCP) THEN
                TRCB_P3_LeakageTestA_ST8A.STATUS.KomunikaciaUkoncena:= TRUE;
                SC_KOM_Server.ResetStep:= TRUE;
                SC_KOM_Server.Step:= 15;
            ELSIF SC_KOM_Server.AlarmTime.Q AND NOT SKTcpClientTrace_1.Status.staSending THEN
                PocetDopytovNaServer:= PocetDopytovNaServer + 1;
				SKTcpClientTrace_1.Cmd.Send:= FALSE;
				SKTcpClientTrace_1.Cmd.Close:= TRUE;
				SC_KOM_Server.ResetStep:= TRUE;
                SC_KOM_Server.Step:= 14;
            END_IF

        14:
            SC_KOM_Server.StepName:= '14 - Vyziadanie stavu paletky - cakam na opatovny dopyt na server';
            SC_KOM_Server.IdleTime.PT:= T#1s;
            SC_KOM_Server.AlarmTime.PT:= T#10s;
            SC_KOM_Server.IdleTime.IN:= TRUE;

            IF PocetDopytovNaServer < 3 THEN
                IF SC_KOM_Server.IdleTime.Q THEN
                    SC_KOM_Server.ResetStep:= TRUE;
                    SC_KOM_Server.Step:= 10;
                END_IF
            ELSE
                TRCB_P3_LeakageTestA_ST8A.STATUS.KomunikaciaError:= TRUE;
                SC_KOM_Server.ResetStep:= TRUE;
                SC_KOM_Server.Step:= 15;
            END_IF

        15:
            SC_KOM_Server.StepName:= '15 - Vyziadanie stavu paletky - cakam na ukoncenie komunikacie';
            SC_KOM_Server.IdleTime.PT:= T#3s;
            SC_KOM_Server.AlarmTime.PT:= T#10s;

            IF NOT TRCB_P3_LeakageTestA_ST8A.CMD.VyziadajStavPaletky_TYP1 THEN
                SC_KOM_Server.ResetStep:= TRUE;
                SC_KOM_Server.Step:= 0;
            END_IF

        20:
            SC_KOM_Server.StepName:= '20 - Priradenie QR kodu - odoslanie dat na server';
            SC_KOM_Server.IdleTime.PT:= T#3s;
            SC_KOM_Server.AlarmTime.PT:= T#10s;

            TRCB_P3_LeakageTestA_ST8A.INPUTS.TYP_Prikazu:= '3';
            TRCB_P3_LeakageTestA_ST8A.INPUTS.CisloStanice:= 'ST8A';
            TRCB_P3_LeakageTestA_ST8A.INPUTS.CisloPaletky;
            TRCB_P3_LeakageTestA_ST8A.INPUTS.QRkodPowerCP:= Paletka[a].PAR.QRkodPowerCP;
            TRCB_P3_LeakageTestA_ST8A.INPUTS.QRkodFiltra:= '';
            TRCB_P3_LeakageTestA_ST8A.INPUTS.ID_Operatora:= Paletka[a].PAR.ID_Operatora;
            TRCB_P3_LeakageTestA_ST8A.INPUTS.Report:= '';
            TRCB_P3_LeakageTestA_ST8A.INPUTS.StavPaletky:= 'OK';
            SKTcpClientTrace_1.Cmd.Send:= TRUE;

            IF SKTcpClientTrace_1.Cmd.Send AND NOT SKTcpClientTrace_1.Status.staReceived AND NOT SKTcpClientTrace_1.Status.staError THEN
                SC_KOM_Server.ResetStep:= TRUE;
                SC_KOM_Server.Step:= 23;
            END_IF

        23:
            SC_KOM_Server.StepName:= '23 - Priradenie QR kodu - odpoved servera';
            SC_KOM_Server.IdleTime.PT:= T#3s;
            SC_KOM_Server.AlarmTime.PT:= T#20s;
            SC_KOM_Server.AlarmTime.IN:= TRUE;

            IF SKTcpClientTrace_1.Status.staReceived AND
                (TRCB_P3_LeakageTestA_ST8A.OUTPUTS.TYP_Prikazu = TRCB_P3_LeakageTestA_ST8A.INPUTS.TYP_Prikazu) AND
                (TRCB_P3_LeakageTestA_ST8A.OUTPUTS.QRkodPowerCP = TRCB_P3_LeakageTestA_ST8A.INPUTS.QRkodPowerCP) THEN
                TRCB_P3_LeakageTestA_ST8A.STATUS.KomunikaciaUkoncena:= TRUE;
                SC_KOM_Server.ResetStep:= TRUE;
                SC_KOM_Server.Step:= 25;
            ELSIF SC_KOM_Server.AlarmTime.Q THEN
                TRCB_P3_LeakageTestA_ST8A.STATUS.KomunikaciaError:= TRUE;
                SC_KOM_Server.ResetStep:= TRUE;
                SC_KOM_Server.Step:= 25;
            END_IF

        25:
            SC_KOM_Server.StepName:= '25 - Vyziadanie stavu paletky - cakam na ukoncenie komunikacie';
            SC_KOM_Server.IdleTime.PT:= T#3s;
            SC_KOM_Server.AlarmTime.PT:= T#10s;

            IF NOT TRCB_P3_LeakageTestA_ST8A.CMD.PriradQRkodFiltra_TYP3 THEN
                SC_KOM_Server.ResetStep:= TRUE;
                SC_KOM_Server.Step:= 0;
            END_IF

        30:
            SC_KOM_Server.StepName:= '30 - Vyziadanie serioveho cisla - odoslanie dat na server';
            SC_KOM_Server.IdleTime.PT:= T#3s;
            SC_KOM_Server.AlarmTime.PT:= T#10s;

            TRCB_P3_LeakageTestA_ST8A.INPUTS.TYP_Prikazu:= '0';
            TRCB_P3_LeakageTestA_ST8A.INPUTS.CisloStanice:= 'ST8A';
            TRCB_P3_LeakageTestA_ST8A.INPUTS.CisloPaletky;
            TRCB_P3_LeakageTestA_ST8A.INPUTS.QRkodPowerCP:= '';
            TRCB_P3_LeakageTestA_ST8A.INPUTS.QRkodFiltra:= '';
            TRCB_P3_LeakageTestA_ST8A.INPUTS.ID_Operatora:= 'E2';
            TRCB_P3_LeakageTestA_ST8A.INPUTS.Report:= '';
            TRCB_P3_LeakageTestA_ST8A.INPUTS.StavPaletky:= 'OK';
            SKTcpClientTrace_1.Cmd.Send:= TRUE;

            IF SKTcpClientTrace_1.Cmd.Send AND NOT SKTcpClientTrace_1.Status.staReceived AND NOT SKTcpClientTrace_1.Status.staError THEN
                SC_KOM_Server.ResetStep:= TRUE;
                SC_KOM_Server.Step:= 33;
            END_IF

        33:
            SC_KOM_Server.StepName:= '33 - Vyziadanie serioveho cisla - odpoved servera';
            SC_KOM_Server.IdleTime.PT:= T#3s;
            SC_KOM_Server.AlarmTime.PT:= T#20s;
            SC_KOM_Server.AlarmTime.IN:= TRUE;

            IF SKTcpClientTrace_1.Status.staReceived AND
                (TRCB_P3_LeakageTestA_ST8A.OUTPUTS.TYP_Prikazu = TRCB_P3_LeakageTestA_ST8A.INPUTS.TYP_Prikazu) THEN
                TRCB_P3_LeakageTestA_ST8A.STATUS.KomunikaciaUkoncena:= TRUE;
                SC_KOM_Server.ResetStep:= TRUE;
                SC_KOM_Server.Step:= 35;
            ELSIF SC_KOM_Server.AlarmTime.Q THEN
                TRCB_P3_LeakageTestA_ST8A.STATUS.KomunikaciaError:= TRUE;
                SC_KOM_Server.ResetStep:= TRUE;
                SC_KOM_Server.Step:= 35;
            END_IF

        35:
            SC_KOM_Server.StepName:= '35 - Vyziadanie serioveho cisla - cakam na ukoncenie komunikacie';
            SC_KOM_Server.IdleTime.PT:= T#3s;
            SC_KOM_Server.AlarmTime.PT:= T#10s;

            IF NOT TRCB_P3_LeakageTestA_ST8A.CMD.VyziadajCisloEtikety_TYP0 THEN
                SC_KOM_Server.ResetStep:= TRUE;
                SC_KOM_Server.Step:= 0;
            END_IF

        40:
            SC_KOM_Server.StepName:= '40 - Odoslanie stavu paletky - odoslanie dat na server';
            SC_KOM_Server.IdleTime.PT:= T#3s;
            SC_KOM_Server.AlarmTime.PT:= T#20s;
            SC_KOM_Server.AlarmTime.IN:= TRUE;

            //Vytvorenie spravy pre report//
            IF NOT SC_KOM_Server.Switch1 THEN
                brsmemset(ADR(Report),0,SIZEOF(Report));
                brsmemset(ADR(TRCB_P3_LeakageTestA_ST8A.INPUTS.Report), 0, SIZEOF(TRCB_P3_LeakageTestA_ST8A.INPUTS.Report));

				//Čas plnenia//
                Report[0].PoradoveCislo:= '1';
                Report[0].Popis:= 'StanicaA_CasPlnenia';
                Report[0].FormatHodnoty:= '1';
                Report[0].Tolerancia_MIN_Hodnota:= '';
                Report[0].Tolerancia_MAX_Hodnota:= '';
                Report[0].Nominal:= '';
                Report[0].Tolerancia_MIN_Jednotky:= '';
                Report[0].Tolerancia_MAX_Jednotky:= '';
                Report[0].NameranaHodnota:= Reports.LeakageTest.CasPlnenia.StanicaA;
                Report[0].NameranaHodnota_Jednotky:= 's';
                Report[0].VyslednyResult:= Reports.LeakageTest.VyslednyReport.StanicaA;
                SKTcpClientNewCsvEntry(Report[0].PoradoveCislo,Report[0].Popis,Report[0].FormatHodnoty,Report[0].Tolerancia_MIN_Hodnota,Report[0].Tolerancia_MAX_Hodnota,Report[0].Nominal,Report[0].Tolerancia_MIN_Jednotky,Report[0].Tolerancia_MAX_Jednotky,Report[0].NameranaHodnota,Report[0].NameranaHodnota_Jednotky,Report[0].VyslednyResult, ADR(TRCB_P3_LeakageTestA_ST8A.INPUTS.Report));

                //Čas stabilizacie//
                Report[1].PoradoveCislo:= '2';
                Report[1].Popis:= 'StanicaA_CasStabilizacie';
                Report[1].FormatHodnoty:= '1';
                Report[1].Tolerancia_MIN_Hodnota:= '';
                Report[1].Tolerancia_MAX_Hodnota:= '';
                Report[1].Nominal:= '';
                Report[1].Tolerancia_MIN_Jednotky:= '';
                Report[1].Tolerancia_MAX_Jednotky:= '';
                Report[1].NameranaHodnota:= Reports.LeakageTest.CasStabilizacie.StanicaA;
                Report[1].NameranaHodnota_Jednotky:= 's';
                Report[1].VyslednyResult:= Reports.LeakageTest.VyslednyReport.StanicaA;
                SKTcpClientNewCsvEntry(Report[1].PoradoveCislo,Report[1].Popis,Report[1].FormatHodnoty,Report[1].Tolerancia_MIN_Hodnota,Report[1].Tolerancia_MAX_Hodnota,Report[1].Nominal,Report[1].Tolerancia_MIN_Jednotky,Report[1].Tolerancia_MAX_Jednotky,Report[1].NameranaHodnota,Report[1].NameranaHodnota_Jednotky,Report[1].VyslednyResult, ADR(TRCB_P3_LeakageTestA_ST8A.INPUTS.Report));

                //Tlak plnenia//
                Report[2].PoradoveCislo:= '3';
                Report[2].Popis:= 'StanicaA_TlakPlnenia';
                Report[2].FormatHodnoty:= '1';
                Report[2].Tolerancia_MIN_Hodnota:= '';
                Report[2].Tolerancia_MAX_Hodnota:= '';
                Report[2].Nominal:= '';
                Report[2].Tolerancia_MIN_Jednotky:= '';
                Report[2].Tolerancia_MAX_Jednotky:= '';
                Report[2].NameranaHodnota:= Reports.LeakageTest.TlakPlnenia.StanicaA;
                Report[2].NameranaHodnota_Jednotky:= 'mBar';
                Report[2].VyslednyResult:= Reports.LeakageTest.VyslednyReport.StanicaA;
                SKTcpClientNewCsvEntry(Report[2].PoradoveCislo,Report[2].Popis,Report[2].FormatHodnoty,Report[2].Tolerancia_MIN_Hodnota,Report[2].Tolerancia_MAX_Hodnota,Report[2].Nominal,Report[2].Tolerancia_MIN_Jednotky,Report[2].Tolerancia_MAX_Jednotky,Report[2].NameranaHodnota,Report[2].NameranaHodnota_Jednotky,Report[2].VyslednyResult, ADR(TRCB_P3_LeakageTestA_ST8A.INPUTS.Report));

                //Tlak prítlaku//
                Report[3].PoradoveCislo:= '4';
                Report[3].Popis:= 'StanicaA_TlakPritlaku';
                Report[3].FormatHodnoty:= '1';
                Report[3].Tolerancia_MIN_Hodnota:= Reports.LeakageTest.ToleranciaPritlaku_MIN.StanicaA;
                Report[3].Tolerancia_MAX_Hodnota:= Reports.LeakageTest.ToleranciaPritlaku_MAX.StanicaA;
                Report[3].Nominal:= '';
                Report[3].Tolerancia_MIN_Jednotky:= 'Bar';
                Report[3].Tolerancia_MAX_Jednotky:= 'Bar';
                Report[3].NameranaHodnota:= Reports.LeakageTest.TlakPritlaku.StanicaA;
                Report[3].NameranaHodnota_Jednotky:= 'Bar';
                Report[3].VyslednyResult:= Reports.LeakageTest.VyslednyReport.StanicaA;
                SKTcpClientNewCsvEntry(Report[3].PoradoveCislo,Report[3].Popis,Report[3].FormatHodnoty,Report[3].Tolerancia_MIN_Hodnota,Report[3].Tolerancia_MAX_Hodnota,Report[3].Nominal,Report[3].Tolerancia_MIN_Jednotky,Report[3].Tolerancia_MAX_Jednotky,Report[3].NameranaHodnota,Report[3].NameranaHodnota_Jednotky,Report[3].VyslednyResult, ADR(TRCB_P3_LeakageTestA_ST8A.INPUTS.Report));

                //Tlak úniku//
                Report[4].PoradoveCislo:= '5';
                Report[4].Popis:= 'StanicaA_TlakUniku';
                Report[4].FormatHodnoty:= '1';
                Report[4].Tolerancia_MIN_Hodnota:= Reports.LeakageTest.ToleranciaTlakUniku_MIN.StanicaA;
                Report[4].Tolerancia_MAX_Hodnota:= Reports.LeakageTest.ToleranciaTlakUniku_MAX.StanicaA;
                Report[4].Nominal:= '';
                Report[4].Tolerancia_MIN_Jednotky:= 'Pa';
                Report[4].Tolerancia_MAX_Jednotky:= 'Pa';
                Report[4].NameranaHodnota:= Reports.LeakageTest.TlakUniku.StanicaA;
                Report[4].NameranaHodnota_Jednotky:= 'Pa';
                Report[4].VyslednyResult:= Reports.LeakageTest.VyslednyReport.StanicaA;
                SKTcpClientNewCsvEntry(Report[4].PoradoveCislo,Report[4].Popis,Report[4].FormatHodnoty,Report[4].Tolerancia_MIN_Hodnota,Report[4].Tolerancia_MAX_Hodnota,Report[4].Nominal,Report[4].Tolerancia_MIN_Jednotky,Report[4].Tolerancia_MAX_Jednotky,Report[4].NameranaHodnota,Report[4].NameranaHodnota_Jednotky,Report[4].VyslednyResult, ADR(TRCB_P3_LeakageTestA_ST8A.INPUTS.Report));

                //Tolerancia//
                Report[5].PoradoveCislo:= '6';
                Report[5].Popis:= 'StanicaA_Tolerancia';
                Report[5].FormatHodnoty:= '1';
                Report[5].Tolerancia_MIN_Hodnota:= '';
                Report[5].Tolerancia_MAX_Hodnota:= '';
                Report[5].Nominal:= '';
                Report[5].Tolerancia_MIN_Jednotky:= '';
                Report[5].Tolerancia_MAX_Jednotky:= '';
                Report[5].NameranaHodnota:= Reports.LeakageTest.Tolerancia.StanicaA;
                Report[5].NameranaHodnota_Jednotky:= 'Pa';
                Report[5].VyslednyResult:= Reports.LeakageTest.VyslednyReport.StanicaA;
                SKTcpClientNewCsvEntry(Report[5].PoradoveCislo,Report[5].Popis,Report[5].FormatHodnoty,Report[5].Tolerancia_MIN_Hodnota,Report[5].Tolerancia_MAX_Hodnota,Report[5].Nominal,Report[5].Tolerancia_MIN_Jednotky,Report[5].Tolerancia_MAX_Jednotky,Report[5].NameranaHodnota,Report[5].NameranaHodnota_Jednotky,Report[5].VyslednyResult, ADR(TRCB_P3_LeakageTestA_ST8A.INPUTS.Report));

                SC_KOM_Server.Switch1:= TRUE;
            END_IF

			TRCB_P3_LeakageTestA_ST8A.INPUTS.CisloPaletky:= 'Pal';
			brsstrcat(ADR(TRCB_P3_LeakageTestA_ST8A.INPUTS.CisloPaletky), ADR(P3_LeakageTestA.PAR.CisloPaletky_STRING));

            TRCB_P3_LeakageTestA_ST8A.INPUTS.TYP_Prikazu:= '2';
            TRCB_P3_LeakageTestA_ST8A.INPUTS.CisloStanice:= 'ST8A';
            TRCB_P3_LeakageTestA_ST8A.INPUTS.QRkodPowerCP:= Paletka[a].PAR.QRkodPowerCP;
            TRCB_P3_LeakageTestA_ST8A.INPUTS.QRkodFiltra:= '';
            TRCB_P3_LeakageTestA_ST8A.INPUTS.ID_Operatora:= Paletka[a].PAR.ID_Operatora;
            TRCB_P3_LeakageTestA_ST8A.INPUTS.StavPaletky:= Paletka[a].PAR.StavPowerCP;

			IF SKTcpClientTrace_1.Status.staReadyToSend AND NOT SKTcpClientTrace_1.Cmd.Close THEN
				TRCB_P3_LeakageTestA_ST8A.OUTPUTS.TYP_Prikazu:= '';
				SKTcpClientTrace_1.Cmd.Send:= TRUE;
				SC_KOM_Server.ResetStep:= TRUE;
				SC_KOM_Server.Step:= 43;
			END_IF

        43:
            SC_KOM_Server.StepName:= '43 - Odoslanie stavu paletky - odpoved servera';
			SC_KOM_Server.IdleTime.PT:= T#3s;
            SC_KOM_Server.AlarmTime.PT:= T#7s;
            SC_KOM_Server.AlarmTime.IN:= TRUE;

            IF SKTcpClientTrace_1.Status.staReceived AND
                (TRCB_P3_LeakageTestA_ST8A.OUTPUTS.TYP_Prikazu = TRCB_P3_LeakageTestA_ST8A.INPUTS.TYP_Prikazu) AND
                (TRCB_P3_LeakageTestA_ST8A.OUTPUTS.QRkodPowerCP = TRCB_P3_LeakageTestA_ST8A.INPUTS.QRkodPowerCP) THEN
                TRCB_P3_LeakageTestA_ST8A.STATUS.KomunikaciaUkoncena:= TRUE;
                SC_KOM_Server.ResetStep:= TRUE;
                SC_KOM_Server.Step:= 45;
            ELSIF SC_KOM_Server.AlarmTime.Q AND NOT SKTcpClientTrace_1.Status.staSending THEN
                PocetDopytovNaServer:= PocetDopytovNaServer + 1;
				SKTcpClientTrace_1.Cmd.Send:= FALSE;
				SKTcpClientTrace_1.Cmd.Close:= TRUE;
				SC_KOM_Server.ResetStep:= TRUE;
                SC_KOM_Server.Step:= 44;
            END_IF

        44:
            SC_KOM_Server.StepName:= '44 - Odoslanie stavu paletky - cakam na opatovny dopyt na server';
            SC_KOM_Server.IdleTime.PT:= T#1s;
            SC_KOM_Server.AlarmTime.PT:= T#10s;
            SC_KOM_Server.IdleTime.IN:= TRUE;
            SKTcpClientTrace_1.Cmd.Send:= FALSE;

            IF PocetDopytovNaServer < 3 THEN
                IF SC_KOM_Server.IdleTime.Q THEN
                    SC_KOM_Server.ResetStep:= TRUE;
                    SC_KOM_Server.Step:= 40;
                END_IF
            ELSE
                TRCB_P3_LeakageTestA_ST8A.STATUS.KomunikaciaError:= TRUE;
                SC_KOM_Server.ResetStep:= TRUE;
                SC_KOM_Server.Step:= 45;
            END_IF

        45:
            SC_KOM_Server.StepName:= '45 - Odoslanie stavu paletky - cakam na ukoncenie komunikacie';
            SC_KOM_Server.IdleTime.PT:= T#3s;
            SC_KOM_Server.AlarmTime.PT:= T#10s;

            IF NOT TRCB_P3_LeakageTestA_ST8A.CMD.OdosliStavPaletky_TYP2 THEN
                SC_KOM_Server.ResetStep:= TRUE;
                SC_KOM_Server.Step:= 0;
            END_IF

		50:
			SC_KOM_Server.StepName:= '50 - Vyziadanie stavu Panatrace - odoslanie dat na server';
			SC_KOM_Server.IdleTime.PT:= T#3s;
			SC_KOM_Server.AlarmTime.PT:= T#10s;
			SC_KOM_Server.AlarmTime.IN:= TRUE;

			TRCB_P3_LeakageTestA_ST8A.INPUTS.TYP_Prikazu:= '4';
			TRCB_P3_LeakageTestA_ST8A.INPUTS.CisloStanice:= 'ST8A';
			TRCB_P3_LeakageTestA_ST8A.INPUTS.CisloPaletky:= '';
			TRCB_P3_LeakageTestA_ST8A.INPUTS.QRkodPowerCP:= '';
			TRCB_P3_LeakageTestA_ST8A.INPUTS.QRkodFiltra:= '';
			TRCB_P3_LeakageTestA_ST8A.INPUTS.ID_Operatora:= '';
			TRCB_P3_LeakageTestA_ST8A.INPUTS.Report:= '';
			TRCB_P3_LeakageTestA_ST8A.INPUTS.StavPaletky:= '';

			IF SKTcpClientTrace_1.Status.staReadyToSend AND NOT SKTcpClientTrace_1.Cmd.Close THEN
				TRCB_P3_LeakageTestA_ST8A.OUTPUTS.TYP_Prikazu:= '';
				SKTcpClientTrace_1.Cmd.Send:= TRUE;
				SC_KOM_Server.ResetStep:= TRUE;
				SC_KOM_Server.Step:= 53;
			END_IF

		53:
			SC_KOM_Server.StepName:= '53 - Vyziadanie stavu paletky - odpoved servera';
			SC_KOM_Server.IdleTime.PT:= T#30s;
			SC_KOM_Server.AlarmTime.PT:= T#7s;
			SC_KOM_Server.AlarmTime.IN:= TRUE;

			IF SKTcpClientTrace_1.Status.staReceived AND TRCB_P3_LeakageTestA_ST8A.OUTPUTS.TYP_Prikazu = TRCB_P3_LeakageTestA_ST8A.INPUTS.TYP_Prikazu THEN
				TRCB_P3_LeakageTestA_ST8A.STATUS.KomunikaciaUkoncena:= TRUE;
				SC_KOM_Server.ResetStep:= TRUE;
				SC_KOM_Server.Step:= 55;
			ELSIF SC_KOM_Server.AlarmTime.Q AND NOT SKTcpClientTrace_1.Status.staSending THEN
				PocetDopytovNaServer:= PocetDopytovNaServer + 1;
				SKTcpClientTrace_1.Cmd.Send:= FALSE;
				SKTcpClientTrace_1.Cmd.Close:= TRUE;
				SC_KOM_Server.ResetStep:= TRUE;
				SC_KOM_Server.Step:= 54;
			END_IF

		54:
			SC_KOM_Server.StepName:= '54 - Vyziadanie stavu paletky - cakam na opatovny dopyt na server';
			SC_KOM_Server.IdleTime.PT:= T#1s;
			SC_KOM_Server.AlarmTime.PT:= T#10s;
			SC_KOM_Server.IdleTime.IN:= TRUE;

			IF PocetDopytovNaServer < 3 THEN
				IF SC_KOM_Server.IdleTime.Q THEN
					SC_KOM_Server.ResetStep:= TRUE;
					SC_KOM_Server.Step:= 50;
				END_IF
			ELSE
				TRCB_P3_LeakageTestA_ST8A.STATUS.KomunikaciaError:= TRUE;
				SC_KOM_Server.ResetStep:= TRUE;
				SC_KOM_Server.Step:= 55;
			END_IF

		55:
			SC_KOM_Server.StepName:= '55 - Vyziadanie stavu paletky - cakam na ukoncenie komunikacie';
			SC_KOM_Server.IdleTime.PT:= T#3s;
			SC_KOM_Server.AlarmTime.PT:= T#10s;

			IF NOT TRCB_P3_LeakageTestA_ST8A.CMD.VyziadajStavPanatrace_TYP4 THEN
				SC_KOM_Server.ResetStep:= TRUE;
				SC_KOM_Server.Step:= 0;
			END_IF

    END_CASE

END_PROGRAM

PROGRAM _EXIT
	(* Insert code here *)

END_PROGRAM
```

#### Types.typ - Local data types
```iecst
TYPE
	Report_typ : 	STRUCT
		PoradoveCislo : STRING[2]; (*IDstep - Poradové čislo reportu*)
		Popis : STRING[100]; (*Description - Popis*)
		FormatHodnoty : STRING[2]; (*TypValue - Format zaslané hodnoty  1- Číslo, 2 - Znak*)
		Tolerancia_MIN_Hodnota : STRING[10]; (*MinTol - Minimálna tolerancia meranej veličiny*)
		Tolerancia_MAX_Hodnota : STRING[10]; (*MaxTol - Maximálna tolerancia meranej veličiny*)
		Nominal : STRING[10]; (*Nom - Ak jezvolený formát string tak tu zadáme OK inak je prazdna*)
		Tolerancia_MIN_Jednotky : STRING[10]; (*MinEle - Jednotky minimálnej tolerancie veličiny*)
		Tolerancia_MAX_Jednotky : STRING[10]; (*MaxEle - Jednotky maximálnej tolerancie veličiny*)
		NameranaHodnota : STRING[10]; (*Value - Namerana hodnota veličiny, ak su kamery tak bude hodnota OK alebo NG*)
		NameranaHodnota_Jednotky : STRING[10]; (*ValEle - Jednotky nameranej veličiny*)
		VyslednyResult : STRING[5]; (*Result - Výsledný result  PASS, FAIL, SKIP*)
	END_STRUCT;
END_TYPE
```

#### Variables.var - Local variables
```iecst
VAR
	SC_KOM_Server : SequenceControlTyp;
	SKTcpClientTrace_1 : SKTcpClientTrace;
	a : USINT;
	Report : ARRAY[0..50] OF Report_typ;
	PocetDopytovNaServer : USINT;
END_VAR
```

### Program Logical/TracebilitySystem/P3_LeakageTestB_ST8B (IEC)

#### Main.st - Init, cyclic, exit code
```iecst
PROGRAM _INIT
	(* Insert code here *)
	SKTcpClientTrace_1.Params.IPportClient := 21001;
	SKTcpClientTrace_1.Cmd.LoggerOn:= FALSE;
END_PROGRAM

PROGRAM _CYCLIC

	//Priradenie indexu paletky//
    a:= P3_LeakageTestB.PAR.CisloPaletky;
	P3_LeakageTestB.PAR.CisloPaletky_STRING:= USINT_TO_STRING(a);

    //Parametre komunikácie//
    memcpy(ADR(SKTcpClientTrace_1.Params.IPaddrServ),ADR('192.168.128.250'),SIZEOF('192.168.128.250'));

    SKTcpClientTrace_1.Params.IPportServ := 12000;

	SKTcpClientTrace_1.pDevice := ADR('HDD_LOGGER');
	SKTcpClientTrace_1.pFile := ADR('logger_sktcpclienttrace_8B.log');
    SKTcpClientTrace_1();

    //Parametre komunikácie//
    //Vstupy pre server//
    SKTcpClientTrace_1.Params.Packet.type := TRCB_P3_LeakageTestB_ST8B.INPUTS.TYP_Prikazu;
    SKTcpClientTrace_1.Params.Packet.workplace := TRCB_P3_LeakageTestB_ST8B.INPUTS.CisloStanice;
    SKTcpClientTrace_1.Params.Packet.rfid := TRCB_P3_LeakageTestB_ST8B.INPUTS.CisloPaletky;
    SKTcpClientTrace_1.Params.Packet.master := TRCB_P3_LeakageTestB_ST8B.INPUTS.QRkodPowerCP;
    SKTcpClientTrace_1.Params.Packet.dps1:= TRCB_P3_LeakageTestB_ST8B.INPUTS.QRkodFiltra;
    SKTcpClientTrace_1.Params.Packet.dps2:= '';
    SKTcpClientTrace_1.Params.Packet.dps3:= '';
    SKTcpClientTrace_1.Params.Packet.dps4:= '';
    SKTcpClientTrace_1.Params.Packet.dps5:= '';
    SKTcpClientTrace_1.Params.Packet.operator_id := TRCB_P3_LeakageTestB_ST8B.INPUTS.ID_Operatora;
    SKTcpClientTrace_1.Params.Packet.data_report:= TRCB_P3_LeakageTestB_ST8B.INPUTS.Report;
    SKTcpClientTrace_1.Params.Packet.result := TRCB_P3_LeakageTestB_ST8B.INPUTS.StavPaletky;

    //Výstupy zo servera//
    TRCB_P3_LeakageTestB_ST8B.OUTPUTS.TYP_Prikazu:= SKTcpClientTrace_1.Internal.Splitter.out[1];
    TRCB_P3_LeakageTestB_ST8B.OUTPUTS.CisloStanice:= SKTcpClientTrace_1.Internal.Splitter.out[2];
    TRCB_P3_LeakageTestB_ST8B.OUTPUTS.CisloPaletky:= SKTcpClientTrace_1.Internal.Splitter.out[3];
    IF TRCB_P3_LeakageTestB_ST8B.INPUTS.TYP_Prikazu = '0' THEN
        TRCB_P3_LeakageTestB_ST8B.OUTPUTS.CisloEtikety:= SKTcpClientTrace_1.Internal.Splitter.out[4];
    ELSE
        TRCB_P3_LeakageTestB_ST8B.OUTPUTS.QRkodPowerCP:= SKTcpClientTrace_1.Internal.Splitter.out[4];
    END_IF
    TRCB_P3_LeakageTestB_ST8B.OUTPUTS.QRkodFiltra:= SKTcpClientTrace_1.Internal.Splitter.out[5];
    TRCB_P3_LeakageTestB_ST8B.OUTPUTS.ID_Operatora:= SKTcpClientTrace_1.Internal.Splitter.out[10];
    TRCB_P3_LeakageTestB_ST8B.OUTPUTS.DruhCinnostiNaPaletke:= SKTcpClientTrace_1.Internal.Splitter.out[11];
    TRCB_P3_LeakageTestB_ST8B.OUTPUTS.PovolenieCinnostiNaPaletke:= SKTcpClientTrace_1.Internal.Splitter.out[12];

    //Volanie funkcie SequenceControl//
    SequenceControl(SC:= SC_KOM_Server);

    CASE SC_KOM_Server.Step OF

        0:
            SC_KOM_Server.StepName:= '0 - Nulovanie';
            SKTcpClientTrace_1.Cmd.Send:= FALSE;
            TRCB_P3_LeakageTestB_ST8B.CMD.VyziadajStavPaletky_TYP1:= FALSE;
            TRCB_P3_LeakageTestB_ST8B.CMD.PriradQRkodFiltra_TYP3:= FALSE;
            TRCB_P3_LeakageTestB_ST8B.CMD.VyziadajCisloEtikety_TYP0:= FALSE;
			TRCB_P3_LeakageTestB_ST8B.CMD.OdosliStavPaletky_TYP2:= FALSE;
			TRCB_P3_LeakageTestB_ST8B.CMD.VyziadajStavPanatrace_TYP4:= FALSE;
            TRCB_P3_LeakageTestB_ST8B.STATUS.KomunikaciaUkoncena:= FALSE;
			TRCB_P3_LeakageTestB_ST8B.STATUS.KomunikaciaError:= FALSE;
			TRCB_P3_LeakageTestB_ST8B.STATUS.KOM_READY:= FALSE;
            PocetDopytovNaServer:= 0;

            IF SKTcpClientTrace_1.Internal.Step = 0 THEN
                SKTcpClientTrace_1.Enable:= TRUE;
                SC_KOM_Server.ResetStep:= TRUE;
                SC_KOM_Server.Step:= 1;
            ELSIF SKTcpClientTrace_1.Internal.Step = 15 THEN
                SKTcpClientTrace_1.Enable:= TRUE;
                SC_KOM_Server.ResetStep:= TRUE;
                SC_KOM_Server.Step:= 1;
            ELSE
                SKTcpClientTrace_1.Enable:= FALSE;
            END_IF

        1:
            SC_KOM_Server.StepName:= '1 - Rozhodnutie o cinnosti';
            TRCB_P3_LeakageTestB_ST8B.STATUS.KOM_READY:= TRUE;
			IF TRCB_P3_LeakageTestB_ST8B.CMD.VyziadajStavPaletky_TYP1 THEN
                TRCB_P3_LeakageTestB_ST8B.STATUS.KOM_READY:= FALSE;
				SC_KOM_Server.Step:= 10;
            ELSIF TRCB_P3_LeakageTestB_ST8B.CMD.PriradQRkodFiltra_TYP3 THEN
                TRCB_P3_LeakageTestB_ST8B.STATUS.KOM_READY:= FALSE;
				SC_KOM_Server.Step:= 20;
            ELSIF TRCB_P3_LeakageTestB_ST8B.CMD.VyziadajCisloEtikety_TYP0 THEN
                TRCB_P3_LeakageTestB_ST8B.STATUS.KOM_READY:= FALSE;
				SC_KOM_Server.Step:= 30;
            ELSIF TRCB_P3_LeakageTestB_ST8B.CMD.OdosliStavPaletky_TYP2 THEN
				TRCB_P3_LeakageTestB_ST8B.STATUS.KOM_READY:= FALSE;
				SC_KOM_Server.Step:= 40;
			ELSIF TRCB_P3_LeakageTestB_ST8B.CMD.VyziadajStavPanatrace_TYP4 THEN
				TRCB_P3_LeakageTestB_ST8B.STATUS.KOM_READY:= FALSE;
				SC_KOM_Server.Step:= 50;
            END_IF

        10:
            SC_KOM_Server.StepName:= '10 - Vyziadanie stavu paletky - odoslanie dat na server';
            SC_KOM_Server.IdleTime.PT:= T#3s;
            SC_KOM_Server.AlarmTime.PT:= T#5s;
            SC_KOM_Server.AlarmTime.IN:= TRUE;

			TRCB_P3_LeakageTestB_ST8B.INPUTS.CisloPaletky:= 'Pal';
			brsstrcat(ADR(TRCB_P3_LeakageTestB_ST8B.INPUTS.CisloPaletky), ADR(P3_LeakageTestB.PAR.CisloPaletky_STRING));

            TRCB_P3_LeakageTestB_ST8B.INPUTS.TYP_Prikazu:= '1';
            TRCB_P3_LeakageTestB_ST8B.INPUTS.CisloStanice:= 'ST8B';
            TRCB_P3_LeakageTestB_ST8B.INPUTS.QRkodPowerCP:= Paletka[a].PAR.QRkodPowerCP;
            TRCB_P3_LeakageTestB_ST8B.INPUTS.QRkodFiltra:= '';
            TRCB_P3_LeakageTestB_ST8B.INPUTS.ID_Operatora:= Paletka[a].PAR.ID_Operatora;
            TRCB_P3_LeakageTestB_ST8B.INPUTS.Report:= '';
            TRCB_P3_LeakageTestB_ST8B.INPUTS.StavPaletky:= 'OK';

			IF SKTcpClientTrace_1.Status.staReadyToSend AND NOT SKTcpClientTrace_1.Cmd.Close THEN
				TRCB_P3_LeakageTestB_ST8B.OUTPUTS.TYP_Prikazu:= '';
				SKTcpClientTrace_1.Cmd.Send:= TRUE;
				SC_KOM_Server.ResetStep:= TRUE;
				SC_KOM_Server.Step:= 13;
			END_IF

		13:
            SC_KOM_Server.StepName:= '13 - Vyziadanie stavu paletky - odpoved servera';
            SC_KOM_Server.IdleTime.PT:= T#3s;
            SC_KOM_Server.AlarmTime.PT:= T#7s;
            SC_KOM_Server.AlarmTime.IN:= TRUE;

            IF SKTcpClientTrace_1.Status.staReceived AND
                (TRCB_P3_LeakageTestB_ST8B.OUTPUTS.TYP_Prikazu = TRCB_P3_LeakageTestB_ST8B.INPUTS.TYP_Prikazu) AND
                (TRCB_P3_LeakageTestB_ST8B.OUTPUTS.QRkodPowerCP = TRCB_P3_LeakageTestB_ST8B.INPUTS.QRkodPowerCP) THEN
                TRCB_P3_LeakageTestB_ST8B.STATUS.KomunikaciaUkoncena:= TRUE;
                SC_KOM_Server.ResetStep:= TRUE;
                SC_KOM_Server.Step:= 15;
            ELSIF SC_KOM_Server.AlarmTime.Q AND NOT SKTcpClientTrace_1.Status.staSending THEN
                PocetDopytovNaServer:= PocetDopytovNaServer + 1;
				SKTcpClientTrace_1.Cmd.Send:= FALSE;
				SKTcpClientTrace_1.Cmd.Close:= TRUE;
				SC_KOM_Server.ResetStep:= TRUE;
                SC_KOM_Server.Step:= 14;
            END_IF

        14:
            SC_KOM_Server.StepName:= '14 - Vyziadanie stavu paletky - cakam na opatovny dopyt na server';
            SC_KOM_Server.IdleTime.PT:= T#1s;
            SC_KOM_Server.AlarmTime.PT:= T#10s;
            SC_KOM_Server.IdleTime.IN:= TRUE;

            IF PocetDopytovNaServer < 3 THEN
                IF SC_KOM_Server.IdleTime.Q THEN
                    SC_KOM_Server.ResetStep:= TRUE;
                    SC_KOM_Server.Step:= 10;
                END_IF
            ELSE
                TRCB_P3_LeakageTestB_ST8B.STATUS.KomunikaciaError:= TRUE;
                SC_KOM_Server.ResetStep:= TRUE;
                SC_KOM_Server.Step:= 15;
            END_IF

        15:
            SC_KOM_Server.StepName:= '15 - Vyziadanie stavu paletky - cakam na ukoncenie komunikacie';
            SC_KOM_Server.IdleTime.PT:= T#3s;
            SC_KOM_Server.AlarmTime.PT:= T#10s;

            IF NOT TRCB_P3_LeakageTestB_ST8B.CMD.VyziadajStavPaletky_TYP1 THEN
                SC_KOM_Server.ResetStep:= TRUE;
                SC_KOM_Server.Step:= 0;
            END_IF

        20:
            SC_KOM_Server.StepName:= '20 - Priradenie QR kodu - odoslanie dat na server';
            SC_KOM_Server.IdleTime.PT:= T#3s;
            SC_KOM_Server.AlarmTime.PT:= T#10s;

            TRCB_P3_LeakageTestB_ST8B.INPUTS.TYP_Prikazu:= '3';
            TRCB_P3_LeakageTestB_ST8B.INPUTS.CisloStanice:= 'ST8B';
            TRCB_P3_LeakageTestB_ST8B.INPUTS.CisloPaletky;
            TRCB_P3_LeakageTestB_ST8B.INPUTS.QRkodPowerCP:= Paletka[a].PAR.QRkodPowerCP;
            TRCB_P3_LeakageTestB_ST8B.INPUTS.QRkodFiltra:= '';
            TRCB_P3_LeakageTestB_ST8B.INPUTS.ID_Operatora:= Paletka[a].PAR.ID_Operatora;
            TRCB_P3_LeakageTestB_ST8B.INPUTS.Report:= '';
            TRCB_P3_LeakageTestB_ST8B.INPUTS.StavPaletky:= 'OK';
            SKTcpClientTrace_1.Cmd.Send:= TRUE;

            IF SKTcpClientTrace_1.Cmd.Send AND NOT SKTcpClientTrace_1.Status.staReceived AND NOT SKTcpClientTrace_1.Status.staError THEN
                SC_KOM_Server.ResetStep:= TRUE;
                SC_KOM_Server.Step:= 23;
            END_IF

        23:
            SC_KOM_Server.StepName:= '23 - Priradenie QR kodu - odpoved servera';
            SC_KOM_Server.IdleTime.PT:= T#3s;
            SC_KOM_Server.AlarmTime.PT:= T#20s;
            SC_KOM_Server.AlarmTime.IN:= TRUE;

            IF SKTcpClientTrace_1.Status.staReceived AND
                (TRCB_P3_LeakageTestB_ST8B.OUTPUTS.TYP_Prikazu = TRCB_P3_LeakageTestB_ST8B.INPUTS.TYP_Prikazu) AND
                (TRCB_P3_LeakageTestB_ST8B.OUTPUTS.QRkodPowerCP = TRCB_P3_LeakageTestB_ST8B.INPUTS.QRkodPowerCP) THEN
                TRCB_P3_LeakageTestB_ST8B.STATUS.KomunikaciaUkoncena:= TRUE;
                SC_KOM_Server.ResetStep:= TRUE;
                SC_KOM_Server.Step:= 25;
            ELSIF SC_KOM_Server.AlarmTime.Q THEN
                TRCB_P3_LeakageTestB_ST8B.STATUS.KomunikaciaError:= TRUE;
                SC_KOM_Server.ResetStep:= TRUE;
                SC_KOM_Server.Step:= 25;
            END_IF

        25:
            SC_KOM_Server.StepName:= '25 - Vyziadanie stavu paletky - cakam na ukoncenie komunikacie';
            SC_KOM_Server.IdleTime.PT:= T#3s;
            SC_KOM_Server.AlarmTime.PT:= T#10s;

            IF NOT TRCB_P3_LeakageTestB_ST8B.CMD.PriradQRkodFiltra_TYP3 THEN
                SC_KOM_Server.ResetStep:= TRUE;
                SC_KOM_Server.Step:= 0;
            END_IF

        30:
            SC_KOM_Server.StepName:= '30 - Vyziadanie serioveho cisla - odoslanie dat na server';
            SC_KOM_Server.IdleTime.PT:= T#3s;
            SC_KOM_Server.AlarmTime.PT:= T#10s;

            TRCB_P3_LeakageTestB_ST8B.INPUTS.TYP_Prikazu:= '0';
            TRCB_P3_LeakageTestB_ST8B.INPUTS.CisloStanice:= 'ST8B';
            TRCB_P3_LeakageTestB_ST8B.INPUTS.CisloPaletky;
            TRCB_P3_LeakageTestB_ST8B.INPUTS.QRkodPowerCP:= '';
            TRCB_P3_LeakageTestB_ST8B.INPUTS.QRkodFiltra:= '';
            TRCB_P3_LeakageTestB_ST8B.INPUTS.ID_Operatora:= 'E2';
            TRCB_P3_LeakageTestB_ST8B.INPUTS.Report:= '';
            TRCB_P3_LeakageTestB_ST8B.INPUTS.StavPaletky:= 'OK';
            SKTcpClientTrace_1.Cmd.Send:= TRUE;

            IF SKTcpClientTrace_1.Cmd.Send AND NOT SKTcpClientTrace_1.Status.staReceived AND NOT SKTcpClientTrace_1.Status.staError THEN
                SC_KOM_Server.ResetStep:= TRUE;
                SC_KOM_Server.Step:= 33;
            END_IF

        33:
            SC_KOM_Server.StepName:= '33 - Vyziadanie serioveho cisla - odpoved servera';
            SC_KOM_Server.IdleTime.PT:= T#3s;
            SC_KOM_Server.AlarmTime.PT:= T#20s;
            SC_KOM_Server.AlarmTime.IN:= TRUE;

            IF SKTcpClientTrace_1.Status.staReceived AND
                (TRCB_P3_LeakageTestB_ST8B.OUTPUTS.TYP_Prikazu = TRCB_P3_LeakageTestB_ST8B.INPUTS.TYP_Prikazu) THEN
                TRCB_P3_LeakageTestB_ST8B.STATUS.KomunikaciaUkoncena:= TRUE;
                SC_KOM_Server.ResetStep:= TRUE;
                SC_KOM_Server.Step:= 35;
            ELSIF SC_KOM_Server.AlarmTime.Q THEN
                TRCB_P3_LeakageTestB_ST8B.STATUS.KomunikaciaError:= TRUE;
                SC_KOM_Server.ResetStep:= TRUE;
                SC_KOM_Server.Step:= 35;
            END_IF

        35:
            SC_KOM_Server.StepName:= '35 - Vyziadanie serioveho cisla - cakam na ukoncenie komunikacie';
            SC_KOM_Server.IdleTime.PT:= T#3s;
            SC_KOM_Server.AlarmTime.PT:= T#10s;

            IF NOT TRCB_P3_LeakageTestB_ST8B.CMD.VyziadajCisloEtikety_TYP0 THEN
                SC_KOM_Server.ResetStep:= TRUE;
                SC_KOM_Server.Step:= 0;
            END_IF

        40:
            SC_KOM_Server.StepName:= '40 - Odoslanie stavu paletky - odoslanie dat na server';
            SC_KOM_Server.IdleTime.PT:= T#3s;
            SC_KOM_Server.AlarmTime.PT:= T#20s;
            SC_KOM_Server.AlarmTime.IN:= TRUE;

            //Vytvorenie spravy pre report//
            IF NOT SC_KOM_Server.Switch1 THEN
                brsmemset(ADR(Report),0,SIZEOF(Report));
                brsmemset(ADR(TRCB_P3_LeakageTestB_ST8B.INPUTS.Report), 0, SIZEOF(TRCB_P3_LeakageTestB_ST8B.INPUTS.Report));

				//Čas plnenia//
                Report[0].PoradoveCislo:= '1';
                Report[0].Popis:= 'StanicaB_CasPlnenia';
                Report[0].FormatHodnoty:= '1';
                Report[0].Tolerancia_MIN_Hodnota:= '';
                Report[0].Tolerancia_MAX_Hodnota:= '';
                Report[0].Nominal:= '';
                Report[0].Tolerancia_MIN_Jednotky:= '';
                Report[0].Tolerancia_MAX_Jednotky:= '';
                Report[0].NameranaHodnota:= Reports.LeakageTest.CasPlnenia.StanicaB;
                Report[0].NameranaHodnota_Jednotky:= 's';
                Report[0].VyslednyResult:= Reports.LeakageTest.VyslednyReport.StanicaB;
                SKTcpClientNewCsvEntry(Report[0].PoradoveCislo,Report[0].Popis,Report[0].FormatHodnoty,Report[0].Tolerancia_MIN_Hodnota,Report[0].Tolerancia_MAX_Hodnota,Report[0].Nominal,Report[0].Tolerancia_MIN_Jednotky,Report[0].Tolerancia_MAX_Jednotky,Report[0].NameranaHodnota,Report[0].NameranaHodnota_Jednotky,Report[0].VyslednyResult, ADR(TRCB_P3_LeakageTestB_ST8B.INPUTS.Report));

                //Čas stabilizacie//
                Report[1].PoradoveCislo:= '2';
                Report[1].Popis:= 'StanicaB_CasStabilizacie';
                Report[1].FormatHodnoty:= '1';
                Report[1].Tolerancia_MIN_Hodnota:= '';
                Report[1].Tolerancia_MAX_Hodnota:= '';
                Report[1].Nominal:= '';
                Report[1].Tolerancia_MIN_Jednotky:= '';
                Report[1].Tolerancia_MAX_Jednotky:= '';
                Report[1].NameranaHodnota:= Reports.LeakageTest.CasStabilizacie.StanicaB;
                Report[1].NameranaHodnota_Jednotky:= 's';
                Report[1].VyslednyResult:= Reports.LeakageTest.VyslednyReport.StanicaB;
                SKTcpClientNewCsvEntry(Report[1].PoradoveCislo,Report[1].Popis,Report[1].FormatHodnoty,Report[1].Tolerancia_MIN_Hodnota,Report[1].Tolerancia_MAX_Hodnota,Report[1].Nominal,Report[1].Tolerancia_MIN_Jednotky,Report[1].Tolerancia_MAX_Jednotky,Report[1].NameranaHodnota,Report[1].NameranaHodnota_Jednotky,Report[1].VyslednyResult, ADR(TRCB_P3_LeakageTestB_ST8B.INPUTS.Report));

                //Tlak plnenia//
                Report[2].PoradoveCislo:= '3';
                Report[2].Popis:= 'StanicaB_TlakPlnenia';
                Report[2].FormatHodnoty:= '1';
                Report[2].Tolerancia_MIN_Hodnota:= '';
                Report[2].Tolerancia_MAX_Hodnota:= '';
                Report[2].Nominal:= '';
                Report[2].Tolerancia_MIN_Jednotky:= '';
                Report[2].Tolerancia_MAX_Jednotky:= '';
                Report[2].NameranaHodnota:= Reports.LeakageTest.TlakPlnenia.StanicaB;
                Report[2].NameranaHodnota_Jednotky:= 'mBar';
                Report[2].VyslednyResult:= Reports.LeakageTest.VyslednyReport.StanicaB;
                SKTcpClientNewCsvEntry(Report[2].PoradoveCislo,Report[2].Popis,Report[2].FormatHodnoty,Report[2].Tolerancia_MIN_Hodnota,Report[2].Tolerancia_MAX_Hodnota,Report[2].Nominal,Report[2].Tolerancia_MIN_Jednotky,Report[2].Tolerancia_MAX_Jednotky,Report[2].NameranaHodnota,Report[2].NameranaHodnota_Jednotky,Report[2].VyslednyResult, ADR(TRCB_P3_LeakageTestB_ST8B.INPUTS.Report));

                //Tlak prítlaku//
                Report[3].PoradoveCislo:= '4';
                Report[3].Popis:= 'StanicaB_TlakPritlaku';
                Report[3].FormatHodnoty:= '1';
                Report[3].Tolerancia_MIN_Hodnota:= Reports.LeakageTest.ToleranciaPritlaku_MIN.StanicaB;
                Report[3].Tolerancia_MAX_Hodnota:= Reports.LeakageTest.ToleranciaPritlaku_MAX.StanicaB;
                Report[3].Nominal:= '';
                Report[3].Tolerancia_MIN_Jednotky:= 'Bar';
                Report[3].Tolerancia_MAX_Jednotky:= 'Bar';
                Report[3].NameranaHodnota:= Reports.LeakageTest.TlakPritlaku.StanicaB;
                Report[3].NameranaHodnota_Jednotky:= 'Bar';
                Report[3].VyslednyResult:= Reports.LeakageTest.VyslednyReport.StanicaB;
                SKTcpClientNewCsvEntry(Report[3].PoradoveCislo,Report[3].Popis,Report[3].FormatHodnoty,Report[3].Tolerancia_MIN_Hodnota,Report[3].Tolerancia_MAX_Hodnota,Report[3].Nominal,Report[3].Tolerancia_MIN_Jednotky,Report[3].Tolerancia_MAX_Jednotky,Report[3].NameranaHodnota,Report[3].NameranaHodnota_Jednotky,Report[3].VyslednyResult, ADR(TRCB_P3_LeakageTestB_ST8B.INPUTS.Report));

                //Tlak úniku//
                Report[4].PoradoveCislo:= '5';
                Report[4].Popis:= 'StanicaB_TlakUniku';
                Report[4].FormatHodnoty:= '1';
                Report[4].Tolerancia_MIN_Hodnota:= Reports.LeakageTest.ToleranciaTlakUniku_MIN.StanicaB;
                Report[4].Tolerancia_MAX_Hodnota:= Reports.LeakageTest.ToleranciaTlakUniku_MAX.StanicaB;
                Report[4].Nominal:= '';
                Report[4].Tolerancia_MIN_Jednotky:= 'Pa';
                Report[4].Tolerancia_MAX_Jednotky:= 'Pa';
                Report[4].NameranaHodnota:= Reports.LeakageTest.TlakUniku.StanicaB;
                Report[4].NameranaHodnota_Jednotky:= 'Pa';
                Report[4].VyslednyResult:= Reports.LeakageTest.VyslednyReport.StanicaB;
                SKTcpClientNewCsvEntry(Report[4].PoradoveCislo,Report[4].Popis,Report[4].FormatHodnoty,Report[4].Tolerancia_MIN_Hodnota,Report[4].Tolerancia_MAX_Hodnota,Report[4].Nominal,Report[4].Tolerancia_MIN_Jednotky,Report[4].Tolerancia_MAX_Jednotky,Report[4].NameranaHodnota,Report[4].NameranaHodnota_Jednotky,Report[4].VyslednyResult, ADR(TRCB_P3_LeakageTestB_ST8B.INPUTS.Report));

                //Tolerancia//
                Report[5].PoradoveCislo:= '6';
                Report[5].Popis:= 'StanicaB_Tolerancia';
                Report[5].FormatHodnoty:= '1';
                Report[5].Tolerancia_MIN_Hodnota:= '';
                Report[5].Tolerancia_MAX_Hodnota:= '';
                Report[5].Nominal:= '';
                Report[5].Tolerancia_MIN_Jednotky:= '';
                Report[5].Tolerancia_MAX_Jednotky:= '';
                Report[5].NameranaHodnota:= Reports.LeakageTest.Tolerancia.StanicaB;
                Report[5].NameranaHodnota_Jednotky:= 'Pa';
                Report[5].VyslednyResult:= Reports.LeakageTest.VyslednyReport.StanicaB;
                SKTcpClientNewCsvEntry(Report[5].PoradoveCislo,Report[5].Popis,Report[5].FormatHodnoty,Report[5].Tolerancia_MIN_Hodnota,Report[5].Tolerancia_MAX_Hodnota,Report[5].Nominal,Report[5].Tolerancia_MIN_Jednotky,Report[5].Tolerancia_MAX_Jednotky,Report[5].NameranaHodnota,Report[5].NameranaHodnota_Jednotky,Report[5].VyslednyResult, ADR(TRCB_P3_LeakageTestB_ST8B.INPUTS.Report));

                SC_KOM_Server.Switch1:= TRUE;
            END_IF

			TRCB_P3_LeakageTestB_ST8B.INPUTS.CisloPaletky:= 'Pal';
			brsstrcat(ADR(TRCB_P3_LeakageTestB_ST8B.INPUTS.CisloPaletky), ADR(P3_LeakageTestB.PAR.CisloPaletky_STRING));

            TRCB_P3_LeakageTestB_ST8B.INPUTS.TYP_Prikazu:= '2';
            TRCB_P3_LeakageTestB_ST8B.INPUTS.CisloStanice:= 'ST8B';
            TRCB_P3_LeakageTestB_ST8B.INPUTS.QRkodPowerCP:= Paletka[a].PAR.QRkodPowerCP;
            TRCB_P3_LeakageTestB_ST8B.INPUTS.QRkodFiltra:= '';
            TRCB_P3_LeakageTestB_ST8B.INPUTS.ID_Operatora:= Paletka[a].PAR.ID_Operatora;
            TRCB_P3_LeakageTestB_ST8B.INPUTS.StavPaletky:= Paletka[a].PAR.StavPowerCP;

			IF SKTcpClientTrace_1.Status.staReadyToSend AND NOT SKTcpClientTrace_1.Cmd.Close THEN
				TRCB_P3_LeakageTestB_ST8B.OUTPUTS.TYP_Prikazu:= '';
				SKTcpClientTrace_1.Cmd.Send:= TRUE;
				SC_KOM_Server.ResetStep:= TRUE;
				SC_KOM_Server.Step:= 43;
			END_IF

        43:
            SC_KOM_Server.StepName:= '43 - Odoslanie stavu paletky - odpoved servera';
			SC_KOM_Server.IdleTime.PT:= T#3s;
            SC_KOM_Server.AlarmTime.PT:= T#7s;
            SC_KOM_Server.AlarmTime.IN:= TRUE;

            IF SKTcpClientTrace_1.Status.staReceived AND
                (TRCB_P3_LeakageTestB_ST8B.OUTPUTS.TYP_Prikazu = TRCB_P3_LeakageTestB_ST8B.INPUTS.TYP_Prikazu) AND
                (TRCB_P3_LeakageTestB_ST8B.OUTPUTS.QRkodPowerCP = TRCB_P3_LeakageTestB_ST8B.INPUTS.QRkodPowerCP) THEN
                TRCB_P3_LeakageTestB_ST8B.STATUS.KomunikaciaUkoncena:= TRUE;
                SC_KOM_Server.ResetStep:= TRUE;
                SC_KOM_Server.Step:= 45;
            ELSIF SC_KOM_Server.AlarmTime.Q AND NOT SKTcpClientTrace_1.Status.staSending THEN
                PocetDopytovNaServer:= PocetDopytovNaServer + 1;
				SKTcpClientTrace_1.Cmd.Send:= FALSE;
				SKTcpClientTrace_1.Cmd.Close:= TRUE;
				SC_KOM_Server.ResetStep:= TRUE;
                SC_KOM_Server.Step:= 44;
            END_IF

        44:
            SC_KOM_Server.StepName:= '44 - Odoslanie stavu paletky - cakam na opatovny dopyt na server';
            SC_KOM_Server.IdleTime.PT:= T#1s;
            SC_KOM_Server.AlarmTime.PT:= T#10s;
            SC_KOM_Server.IdleTime.IN:= TRUE;
            SKTcpClientTrace_1.Cmd.Send:= FALSE;

            IF PocetDopytovNaServer < 3 THEN
                IF SC_KOM_Server.IdleTime.Q THEN
                    SC_KOM_Server.ResetStep:= TRUE;
                    SC_KOM_Server.Step:= 40;
                END_IF
            ELSE
                TRCB_P3_LeakageTestB_ST8B.STATUS.KomunikaciaError:= TRUE;
                SC_KOM_Server.ResetStep:= TRUE;
                SC_KOM_Server.Step:= 45;
            END_IF

        45:
            SC_KOM_Server.StepName:= '45 - Odoslanie stavu paletky - cakam na ukoncenie komunikacie';
            SC_KOM_Server.IdleTime.PT:= T#3s;
            SC_KOM_Server.AlarmTime.PT:= T#10s;

            IF NOT TRCB_P3_LeakageTestB_ST8B.CMD.OdosliStavPaletky_TYP2 THEN
                SC_KOM_Server.ResetStep:= TRUE;
                SC_KOM_Server.Step:= 0;
            END_IF

		50:
			SC_KOM_Server.StepName:= '50 - Vyziadanie stavu Panatrace - odoslanie dat na server';
			SC_KOM_Server.IdleTime.PT:= T#3s;
			SC_KOM_Server.AlarmTime.PT:= T#10s;
			SC_KOM_Server.AlarmTime.IN:= TRUE;

			TRCB_P3_LeakageTestB_ST8B.INPUTS.TYP_Prikazu:= '4';
			TRCB_P3_LeakageTestB_ST8B.INPUTS.CisloStanice:= 'ST8B';
			TRCB_P3_LeakageTestB_ST8B.INPUTS.CisloPaletky:= '';
			TRCB_P3_LeakageTestB_ST8B.INPUTS.QRkodPowerCP:= '';
			TRCB_P3_LeakageTestB_ST8B.INPUTS.QRkodFiltra:= '';
			TRCB_P3_LeakageTestB_ST8B.INPUTS.ID_Operatora:= '';
			TRCB_P3_LeakageTestB_ST8B.INPUTS.Report:= '';
			TRCB_P3_LeakageTestB_ST8B.INPUTS.StavPaletky:= '';

			IF SKTcpClientTrace_1.Status.staReadyToSend AND NOT SKTcpClientTrace_1.Cmd.Close THEN
				TRCB_P3_LeakageTestB_ST8B.OUTPUTS.TYP_Prikazu:= '';
				SKTcpClientTrace_1.Cmd.Send:= TRUE;
				SC_KOM_Server.ResetStep:= TRUE;
				SC_KOM_Server.Step:= 53;
			END_IF

		53:
			SC_KOM_Server.StepName:= '53 - Vyziadanie stavu paletky - odpoved servera';
			SC_KOM_Server.IdleTime.PT:= T#30s;
			SC_KOM_Server.AlarmTime.PT:= T#7s;
			SC_KOM_Server.AlarmTime.IN:= TRUE;

			IF SKTcpClientTrace_1.Status.staReceived AND TRCB_P3_LeakageTestB_ST8B.OUTPUTS.TYP_Prikazu = TRCB_P3_LeakageTestB_ST8B.INPUTS.TYP_Prikazu THEN
				TRCB_P3_LeakageTestB_ST8B.STATUS.KomunikaciaUkoncena:= TRUE;
				SC_KOM_Server.ResetStep:= TRUE;
				SC_KOM_Server.Step:= 55;
			ELSIF SC_KOM_Server.AlarmTime.Q AND NOT SKTcpClientTrace_1.Status.staSending THEN
				PocetDopytovNaServer:= PocetDopytovNaServer + 1;
				SKTcpClientTrace_1.Cmd.Send:= FALSE;
				SKTcpClientTrace_1.Cmd.Close:= TRUE;
				SC_KOM_Server.ResetStep:= TRUE;
				SC_KOM_Server.Step:= 54;
			END_IF

		54:
			SC_KOM_Server.StepName:= '54 - Vyziadanie stavu paletky - cakam na opatovny dopyt na server';
			SC_KOM_Server.IdleTime.PT:= T#1s;
			SC_KOM_Server.AlarmTime.PT:= T#10s;
			SC_KOM_Server.IdleTime.IN:= TRUE;

			IF PocetDopytovNaServer < 3 THEN
				IF SC_KOM_Server.IdleTime.Q THEN
					SC_KOM_Server.ResetStep:= TRUE;
					SC_KOM_Server.Step:= 50;
				END_IF
			ELSE
				TRCB_P3_LeakageTestB_ST8B.STATUS.KomunikaciaError:= TRUE;
				SC_KOM_Server.ResetStep:= TRUE;
				SC_KOM_Server.Step:= 55;
			END_IF

		55:
			SC_KOM_Server.StepName:= '55 - Vyziadanie stavu paletky - cakam na ukoncenie komunikacie';
			SC_KOM_Server.IdleTime.PT:= T#3s;
			SC_KOM_Server.AlarmTime.PT:= T#10s;

			IF NOT TRCB_P3_LeakageTestB_ST8B.CMD.VyziadajStavPanatrace_TYP4 THEN
				SC_KOM_Server.ResetStep:= TRUE;
				SC_KOM_Server.Step:= 0;
			END_IF

    END_CASE

END_PROGRAM

PROGRAM _EXIT
	(* Insert code here *)

END_PROGRAM
```

#### Types.typ - Local data types
```iecst
TYPE
	Report_typ : 	STRUCT
		PoradoveCislo : STRING[2]; (*IDstep - Poradové čislo reportu*)
		Popis : STRING[100]; (*Description - Popis*)
		FormatHodnoty : STRING[2]; (*TypValue - Format zaslané hodnoty  1- Číslo, 2 - Znak*)
		Tolerancia_MIN_Hodnota : STRING[10]; (*MinTol - Minimálna tolerancia meranej veličiny*)
		Tolerancia_MAX_Hodnota : STRING[10]; (*MaxTol - Maximálna tolerancia meranej veličiny*)
		Nominal : STRING[10]; (*Nom - Ak jezvolený formát string tak tu zadáme OK inak je prazdna*)
		Tolerancia_MIN_Jednotky : STRING[10]; (*MinEle - Jednotky minimálnej tolerancie veličiny*)
		Tolerancia_MAX_Jednotky : STRING[10]; (*MaxEle - Jednotky maximálnej tolerancie veličiny*)
		NameranaHodnota : STRING[10]; (*Value - Namerana hodnota veličiny, ak su kamery tak bude hodnota OK alebo NG*)
		NameranaHodnota_Jednotky : STRING[10]; (*ValEle - Jednotky nameranej veličiny*)
		VyslednyResult : STRING[5]; (*Result - Výsledný result  PASS, FAIL, SKIP*)
	END_STRUCT;
END_TYPE
```

#### Variables.var - Local variables
```iecst
VAR
	SC_KOM_Server : SequenceControlTyp;
	SKTcpClientTrace_1 : SKTcpClientTrace;
	a : USINT;
	Report : ARRAY[0..50] OF Report_typ;
	PocetDopytovNaServer : USINT;
END_VAR
```

### Program Logical/TracebilitySystem/P4_Etiketovacka_ST9 (IEC)
